// ---- POUs/HydraulicsControl.TcPOU
PROGRAM HydraulicsControl
VAR_INPUT
	// start the hydraulics
	enable:		BOOL := FALSE;
	// reset any hydraulics error
	reset: 		BOOL;
	// manual override to start the suction pump
	suction_manual:	BOOL;
	//manual override to stop the pump
	pump_manual_stop: BOOL;
END_VAR
VAR_OUTPUT
	// status of the brake: is the brake open?
	brake_open:			BOOL;
	// is the brake closed?
	brake_closed:		BOOL;
	// pump is running, but the pressure remains low
	pressure_failure:	BOOL;
	// suction was started, but it is not running
	suction_failure:	BOOL;
	// main pump is running but suction has a timeout
	hydraulics_failure:	BOOL;
	main_pump_failure: BOOL;
	// oil is low
	oil_low:			BOOL;
	// oil is high (unused?)
	oil_high:			BOOL;
	// oil pressure is 25 bars
	oil_pressure_OK:	BOOL;
	// oil is on reserve
	oil_warning:		BOOL;
	// oil filter is dirty
	oil_filter_dirty:	BOOL;
	// oil is below 10°C
	oil_cold:			BOOL;
	// oil is above 50°C
	oil_hot:			BOOL;
	// main pump is running
	pump_running:		BOOL;
	// suction pump is running
	suction_running :	BOOL := FALSE;
	// error condition
	error: 				BOOL;
END_VAR
VAR
	// command to open the brake
	iopen_brake:	BOOL := FALSE;
	// command to open the brake
	iclose_brake: BOOL;
	// monitors the pressure of the pump is running
	pressure_watchdog:	TON;
	// monitors the activation of the suction pump
	suction_watchdog: TON;
	// monitors the activation of the main pump
	main_pump_watchdog:	TON;
	// watch the hydraulics and suction pumps
	hydraulics_watchdog: TON;
	// represents the state of the main pump
	oil_pump_state:		RS;
	// represents the state of the brake
	brake_state: 		RS;
	// wait for the brake to open after pressure has been established
	brake_open_delay:	TON;
	// report brake opend after a short delay
	brake_opened_delay:	TON;
	// error state (set dominant)
	error_state:	SR;
	// trigger for suction pump
	suction_trigger:	SR;
	// timer to shut off hydraulics after break was closed
	hydraulics_off_timer:	TON  := (PT := T#300S);
	off_trigger:	F_TRIG;
	oil_level, last_oil_level:		REAL;
	HydraulicsLog,
	PumpLog,
	ReserveLog,
	oil_low_log,
	FilterLog,
	oil_max_log,
	OverTemperatureLog,
	UnderTemperatureLog,
	SuctionLog,
	HydraulicsFailureLog,
	BrakeClearingWarning,
	BrakeHydraulicsWarning,
	BrakeWarning: FB_EventLog;
	
	// measures the operating cycle of the suction pump
	suction_timer : FB_Timer;
	StatusWord, LastStatus:	UDINT;
END_VAR

(* 
Main control Logic for the Hydraulics system
* power on delay for main pump and suction pump
* start main pump if main control is ready (button pressed or remote)
* start suction pump if maximum in pan is reached
* suction pump runs for 60 seconds
* stop main pump if oil is low
* stop main pump if pressure fails for 10 seconds
*)
oil_low := NOT GVL_Hydraulics.oil_low;
oil_high := NOT GVL_Hydraulics.oil_high;
oil_warning := GVL_Hydraulics.oil_reserve;
oil_pressure_OK := GVL_Hydraulics.oil_pressure_OK;
oil_filter_dirty := NOT GVL_Hydraulics.oilfilter_dirty;
oil_cold := NOT GVL_Hydraulics.oil_undertemperature;
oil_hot := GVL_Hydraulics.oil_overtemperature;
oil_level := F_YREAL(GVL_Hydraulics.oil_level, 0, 16383, 0.0, 5.0);
pump_running := GVL_Hydraulics.pump_running;
suction_running := GVL_Hydraulics.suction_running;

error_state(SET1 := pressure_failure OR	suction_failure OR hydraulics_failure OR oil_low OR main_pump_failure,
			RESET := reset,
			Q1 => error);
// clear reset, if no error present

IF NOT error THEN
	reset := FALSE;
END_IF

oil_pump_state(SET := enable,
				RESET1 := NOT enable OR error OR pump_manual_stop OR GVL_Hydraulics.oilpan_maximum);

GVL_Hydraulics.oil_pump_enable := oil_pump_state.Q1;

(* This section controls the hydraulic brake responsible for azimuth and elevation. 
Especially the elevation is imbalanced if not in the position control loop. 
The brake must only be opened, if the elevation drive is activated concurrently.
*)


// close the brake if the pump is not running	
IF iclose_brake OR NOT pump_running THEN 
	iopen_brake := FALSE;
END_IF

// wait for pressure to build up (hack for oil_pressure_ok)
brake_open_delay(IN := pump_running AND oil_pressure_OK,
				PT := T#3S);
		
brake_state(SET := brake_open_delay.Q AND iopen_brake AND MAIN.brake_clearing,
			RESET1 := GVL_Telescope.azimut_limit_switch 
					  OR iclose_brake 
					  OR NOT pump_running
					  OR NOT MAIN.brake_clearing,
			Q1 => GVL_Telescope.brake_azimuth_eve);

// signal that the brake is open after one second
brake_opened_delay(	IN :=brake_state.Q1, 
					PT := T#1000MS,
					Q => brake_open);

brake_closed := NOT brake_open;
IF brake_closed THEN
	iclose_brake := FALSE;
END_IF
// turn off the hydraulics if the brake is closed and the pump is still running
hydraulics_off_timer(IN := brake_closed AND enable );
off_trigger(CLK := hydraulics_off_timer.Q);

IF hydraulics_off_timer.Q THEN
	enable := FALSE;
END_IF

(* This is the end of the brake control section *)

suction_trigger(SET1 := GVL_Hydraulics.oilpan_maximum OR oil_level>3.7,
				RESET := oil_level<3.0);
GVL_Hydraulics.oil_suction_enable := suction_trigger.Q1 OR suction_manual;					
suction_watchdog(IN := GVL_Hydraulics.oil_suction_enable AND NOT suction_running,
					PT := T#15S,
					Q => suction_failure);
					
pressure_watchdog(IN := GVL_Hydraulics.oil_pump_enable AND 
						NOT oil_pressure_OK,
					PT := T#30S,
				  Q => pressure_failure);
hydraulics_watchdog(IN := pump_running AND NOT suction_running,
						PT := T#140S,
						Q => hydraulics_failure);

main_pump_watchdog(IN := GVL_Hydraulics.oil_pump_enable AND NOT pump_running,
					PT := T#10S,
					Q => main_pump_failure);

StatusWord.0 := oil_low;
StatusWord.1 := oil_high;
StatusWord.2 := oil_warning;
StatusWord.3 := oil_pressure_OK;
StatusWord.4 := oil_filter_dirty;
StatusWord.5 := oil_cold;
StatusWord.6 := oil_hot;
StatusWord.7 := brake_open;
StatusWord.8 := GVL_Main.brake_clearing;
StatusWord.9 := pump_running;
StatusWord.10 := suction_running;
StatusWord.11 := GVL_Hydraulics.oilpan_maximum;
StatusWord.12 := GVL_Hydraulics.oil_pump_enable;
StatusWord.13 := GVL_Hydraulics.oil_suction_enable;
IF ABS(last_oil_level - oil_level) > 0.02 THEN
	StatusWord.15 := TRUE;
	last_oil_level := oil_level;
ELSE
	StatusWord.15 := FALSE;
END_IF

IF StatusWord<>LastStatus THEN // publish new payload every second
	LastStatus := StatusWord;
	MAIN.MQTTClient.Publish('hydraulics', 'base', 'OilLow',			BOOL_TO_STRING(oil_low));
	MAIN.MQTTClient.Publish('hydraulics', 'base', 'OilHigh',		BOOL_TO_STRING(oil_high));
	MAIN.MQTTClient.Publish('hydraulics', 'base', 'OilMaximum',		BOOL_TO_STRING(GVL_Hydraulics.oilpan_maximum));
	MAIN.MQTTClient.Publish('hydraulics', 'base', 'OilReserve',		BOOL_TO_STRING(oil_warning));
	MAIN.MQTTClient.Publish('hydraulics', 'base', 'OilPressureOK', 	BOOL_TO_STRING(oil_pressure_OK));
	MAIN.MQTTClient.Publish('hydraulics', 'base', 'OilFilterDirty',	BOOL_TO_STRING(oil_filter_dirty));
	MAIN.MQTTClient.Publish('hydraulics', 'base', 'OilCold',		BOOL_TO_STRING(oil_cold));
	MAIN.MQTTClient.Publish('hydraulics', 'base', 'OilHot',			BOOL_TO_STRING(oil_Hot));
	MAIN.MQTTClient.Publish('hydraulics', 'base', 'BrakeOpen',		BOOL_TO_STRING(brake_open));
	MAIN.MQTTClient.Publish('hydraulics', 'base', 'BrakeClearing',	BOOL_TO_STRING(GVL_Main.brake_clearing));
	MAIN.MQTTClient.Publish('hydraulics', 'base', 'PumpRunning',	BOOL_TO_STRING(pump_running));
	MAIN.MQTTClient.Publish('hydraulics', 'base', 'SuctionRunning',	BOOL_TO_STRING(suction_running));
	MAIN.MQTTClient.Publish('hydraulics', 'base', 'OilLevel',		REAL_TO_STRING(oil_level));
	MAIN.MQTTClient.Publish('hydraulics', 'base', 'StatusWord',		UDINT_TO_STRING(StatusWord));
END_IF


				  				  
HydraulicsLog(Trigger := pressure_failure OR main_pump_failure,
				Level := ADSLOG_MSGTYPE_ERROR,
				FormatString := 'Main hydraulics pump / pressure: %s',
				OnMessage := 'FAILURE',
				OffMessage := 'OK',
				OffLevel := ADSLOG_MSGTYPE_HINT);

PumpLog(Trigger := pump_running,
				Level := ADSLOG_MSGTYPE_HINT,
				FormatString := 'Main hydraulics pump: %s',
				OnMessage := 'START',
				OffMessage := 'STOP',
				OffLevel := ADSLOG_MSGTYPE_HINT);
	
ReserveLog(Trigger := oil_warning,
			Level := ADSLOG_MSGTYPE_WARN,
			FormatString := 'oil reserve: %s',
			OnMessage := 'LOW',
			OffMessage := 'OK',
			OffLevel := ADSLOG_MSGTYPE_HINT);

oil_low_log(Trigger := oil_low,
				Level := ADSLOG_MSGTYPE_ERROR,
				FormatString := 'oil level: %s',
				OnMessage := 'LOW',
				OffMessage := 'OK',
				OffLevel := ADSLOG_MSGTYPE_HINT);

oil_max_log(Trigger := GVL_Hydraulics.oilpan_maximum,
				Level := ADSLOG_MSGTYPE_ERROR,
				FormatString := 'oil level: %s',
				OnMessage := 'MAXIMUM',
				OffMessage := 'OK',
				OffLevel := ADSLOG_MSGTYPE_HINT);	
				
FilterLog(Trigger := oil_filter_dirty,
				Level := ADSLOG_MSGTYPE_WARN,
				FormatString := 'Hydraulics Filter is %s',
				OnMessage := 'dirty.');

OverTemperatureLog(Trigger := oil_hot,
				Level := ADSLOG_MSGTYPE_WARN,
				FormatString := 'Hydraulics Temperature is %s',
				OnMessage := 'high.');
				
UnderTemperatureLog(Trigger := oil_cold,
				Level := ADSLOG_MSGTYPE_WARN,
				FormatString := 'Hydraulics Temperature is %s',
				OnMessage := 'low.');

SuctionLog(Trigger := suction_failure,
				Level := ADSLOG_MSGTYPE_ERROR,
				FormatString := 'suction pump: %s',
				OnMessage := 'FAILURE',
				OffMessage := 'OK',
				OffLevel := ADSLOG_MSGTYPE_HINT);

HydraulicsFailureLog(Trigger := hydraulics_failure,
				Level := ADSLOG_MSGTYPE_ERROR,
				FormatString := 'suction pump while running main pump: %s',
				OnMessage := 'FAILURE',
				OffMessage := 'OK',
				OffLevel := ADSLOG_MSGTYPE_HINT);
				
BrakeClearingWarning(Trigger := NOT Main.brake_clearing AND iopen_brake,
				Level := ADSLOG_MSGTYPE_WARN,
				FormatString := '%s',
				OnMessage := 'Cannot open brake without brake clearing.');

BrakeWarning(	Trigger := brake_open,
				Level := ADSLOG_MSGTYPE_WARN,
				FormatString := '%s',
				OnMessage := 'Brake is open.',
				OffMessage := 'Brake is closed.');

BrakeHydraulicsWarning(Trigger := NOT enable AND iopen_brake,
				Level := ADSLOG_MSGTYPE_WARN,
				FormatString := '%s',
				OnMessage := 'Cannot open brake without running hydraulics.');

METHOD close_brake : BOOL
VAR_INPUT
END_VAR
// close the brake
iclose_brake := TRUE;

RETURN(brake_closed);
END_METHOD

METHOD open_brake : BOOL
VAR_INPUT
END_VAR
// start the pump
enable := TRUE;
// open the brake
IF oil_pressure_OK THEN
	iopen_brake := TRUE;
END_IF;
RETURN(brake_open);
END_METHOD

END_PROGRAM

// ---- POUs/Functions/F_YREAL.TcPOU
FUNCTION F_YREAL : REAL
VAR_INPUT
	fX:		LREAL;
	fXmin:	REAL := 0.0;
	fXmax:	REAL := 32767.0;
	fYmin, fYmax:	REAL;
END_VAR
VAR
	fgain,
	foffset:	LREAL;
END_VAR

(*
y = mx+b

		    delta X	  fYmax - fYmin
m = fgain = ------- = -------------
			delta Y	  fXmax - fXmin
			
b = foffset = y - m*x = y - fgain*x
					  = fYmin - fgain * fXmin
*)

// y = fgain * x + foffset

IF (fXmax - fXmin) <> 0 THEN

	// Berechnung der Steigung
	fgain := (fYmax - fYmin) / (fXmax - fXmin);
	
	// Berechnung des Offsets
	foffset := fYmin - (fgain * fXmin);
	
	// Berechnung von F_Y

	F_YREAL := LREAL_TO_REAL(fgain * fX + foffset);
	F_YREAL := LIMIT(fYmin, F_YREAL, fYMAX);
END_IF

END_FUNCTION

// ---- POUs/AzimuthElevationControl.TcPOU
PROGRAM AzimuthElevationControl
VAR_INPUT
	// enable the axis and its position control loop
	Enable:		BOOL;
	// reset the axis
	Reset: 		BOOL;
	// decrease azimuth
	left:		BOOL;
	// increase azimuth
	right: 		BOOL;
	// Move azimuth to given position
	MoveAxis:	BOOL;
	// Home the axis
	HomeAxis:	BOOL;
	// enable tracking
	Tracking:	BOOL;
	// position to move the axis to
	position: 	LREAL;
	// set the Velocity of the axis
	velocity:	LREAL;
	// stop the Axis
	StopAxis:	BOOL;
	// diagnostic reset
	bSoEReset:	BOOL;
END_VAR
VAR_OUTPUT
	// error state of the axis
	error: 			BOOL;
	// error ID of the axis
	ErrorID:		UDINT;
	// actual_position of the axis
	act_position:	LREAL;
	// is the axis calibrated
	calibrated:		BOOL;
	// drive is ready
	ready:			BOOL;
	// time to reach target position
	slewtime:		LREAL;
END_VAR
VAR
	AzimuthAxis:		FB_Axis2;
	AzimuthCalibration: MC_SetPosition;
	//fbSoEReset:			FB_SoEReset;
	AzimuthAxisEvent: 	FB_EventLog;
	AzimuthDiagnosticEvent: 	FB_EventLog;
	// delay until commutator angle is measured
	readydelay:			TON;
	HomeDelay:			FB_TONTP;
	TorqueError:		TON := (PT := T#3S);
	azimuth_torque: 	REAL;
	TorqueWarning:		FB_EventLog;
	CalibrationEvent:	FB_Eventlog;
	ReadParameter:		MC_ReadParameter;
	getlastposition:	BOOL := TRUE;
	azimuth_rest_timer:	TON;
	azimuth_at_rest:	BOOL;
	fbSoEReset: 		FB_SoEReset;
	DiagnosticError:	BOOL;
END_VAR
VAR CONSTANT
	// reference position for homing
	// homing_position:		LREAL := 439.0; // was 442 - -21.21 = 463.21; 463 + 24 = 439
	// current position of the calibration cam encoder zero index. Apply an offset here if necessary
	calibration_position:	LREAL :=  208.4983;//208.6273; //208.6073; // 208.7122869;//207.0092; // 208.2342; 
END_VAR
VAR PERSISTENT
	last_position:	LREAL := -1.0;
END_VAR

(* Azimuth Axis control section
Power must be on and brake must be open for the axis to operate
*)

// generate the ready signal after enabling the drive
readydelay(IN :=  AzimuthAxis.Enable, PT := T#3000MS, Q=> ready);

// limit the input position angle
position := LIMIT(0.0, position, 450.0);

// conduct the calibrated signal
calibrated := AzimuthAxis.Calibrated;

IF Calibrated OR Error THEN
	HomeAxis := FALSE;
	getlastposition := FALSE;
END_IF
	
IF HomeAxis THEN
	position := calibration_position;
END_IF

IF HomeDelay.Q THEN
	position := calibration_position;
	MoveAxis := TRUE;
END_IF

// perform a recalibration on the last known position
AzimuthCalibration(
	Axis := GVL_Telescope.AzimuthAxisRef,
	Execute := getlastposition AND last_position>=0.0 AND NOT Calibrated,
	Position := last_position);

IF AzimuthCalibration.Done THEN
	getlastposition := FALSE;
END_IF

IF Calibrated THEN
	last_position := act_position;
END_IF

// enable the azimuth if not moved by the power chain. Sorry for the hack
azimuth_rest_timer(IN := HydraulicsControl.brake_open AND 
				(ABS(GVL_Telescope.AzimuthAxisRef.NcToPlc.ActVelo) < 0.01), PT := T#2S);
// if azimuth at rest or calibrated, allow enabling the azimuth
IF azimuth_rest_timer.Q or calibrated THEN
	azimuth_at_rest := TRUE;
ELSIF HydraulicsControl.brake_closed THEN
	azimuth_at_rest := FALSE;
END_IF
	
// deactivate limit switches on homing
MC_SetAcceptBlockedDriveSignal(
	Axis := GVL_Telescope.AzimuthAxisRef, 
	Enable := HomeAxis);

AzimuthAxis(	
	Enable := 			enable AND azimuth_at_rest AND NOT GVL_Telescope.azimut_limit_switch,
	Reset := 			reset,
	MoveAxis :=			MoveAxis,
	HomeAxis := 		HomeAxis,
	StopAxis :=			StopAxis,
	Tracking :=			Tracking,
	Position := 		position, 
	Velocity :=			velocity,
	Enable_Positive := 	GVL_Telescope.Azimuth_inputs.1 OR HomeAxis,
	Enable_Negative := 	GVL_Telescope.Azimuth_inputs.0,
	Jog_Forward :=		right,
	Jog_Backwards := 	left,
	bCalibrationCam :=	NOT GVL_Telescope.Azimuth_inputs.1,
	ActualPosition => 	act_position,
	Error => 			error,
	ErrorID => 			ErrorID,
	AxisRef :=			GVL_Telescope.AzimuthAxisRef);

IF bSoEReset THEN
	last_position := -1.0;
	fbSoEReset(
		Axis := GVL_Telescope.AzimuthAxisRef,
		Execute := TRUE,
		Timeout := DEFAULT_ADS_TIMEOUT);
 	IF fbSoEReset.Busy THEN
		fbSoEReset(Axis := GVL_Telescope.AzimuthAxisRef, Execute := FALSE);
	ELSE
		bSoEReset := FALSE;
		Reset := TRUE;
	END_IF
END_IF 

IF AzimuthAxis.MoveDone THEN
	MoveAxis := FALSE;
END_IF

IF AzimuthAxis.HomeDone THEN
	HomeAxis := FALSE;
END_IF
	
IF AzimuthAxis.ResetDone THEN
	reset := FALSE;
END_IF

IF AzimuthAxis.StopDone THEN
	StopAxis := FALSE;
END_IF
DiagnosticError := FALSE;
IF GVL_Telescope.Azimuth_diagnostic < 16#D012 AND GVL_Telescope.Azimuth_diagnostic > 16#D014 THEN
	DiagnosticError :=TRUE;
	ErrorID := GVL_Telescope.Azimuth_diagnostic;
END_IF

ReadParameter(	Axis := GVL_Telescope.AzimuthAxisRef, Enable := AzimuthAxis.InMotion, 
				ParameterNumber := MC_AxisParameter.AxisRemainingTimeToGo, 
				ReadMode := E_ReadMode.READMODE_CYCLIC);
IF ReadParameter.Valid THEN
	slewtime := ReadParameter.Value;
END_IF

azimuth_torque := GVL_Telescope.Azimuth_torque / 10.0;
TorqueError(IN := ABS(azimuth_torque) > 50.0);


AzimuthAxisEvent(	
	Trigger := 		Error, 
	Level := 		ADSLOG_MSGTYPE_ERROR,
	FormatString :=	'Azimuth Axis Error: %s',
	OnMessage := 	NCError_TO_STRING(ErrorID));
	
AzimuthDiagnosticEvent(	
	Trigger := 		DiagnosticError,
	Level := 		ADSLOG_MSGTYPE_ERROR,
	FormatString :=	'Azimuth Axis Diagnostic Error: %s',
	OnMessage := 	NCError_TO_STRING(GVL_Telescope.Azimuth_diagnostic));
	
TorqueWarning(	
	Trigger := 		TorqueError.Q, 
	Level := 		ADSLOG_MSGTYPE_WARN,
	FormatString :=	'%s',
	OnMessage := 	'Azimuth torque is high.');
	
CalibrationEvent(
	Trigger := 		Calibrated, 
	Level := 		ADSLOG_MSGTYPE_HINT,
	FormatString :=	'%s',
	OnMessage := 	'Azimuth axis is calibrated.');

END_PROGRAM

// ---- POUs/FunctionBlocks/FB_TONTP.TcPOU
FUNCTION_BLOCK FB_TONTP
VAR_INPUT
	IN :	BOOL;
	 PT1:	TIME := T#1000MS;
	 PT2:	TIME := T#1000MS;
END_VAR
VAR_OUTPUT
	Q:	BOOL;
END_VAR
VAR
	ton:	TON;
	tp:		TP;
END_VAR

ton(IN := IN, PT := PT1);
tp(IN := ton.Q, PT := PT2, Q => Q);

END_FUNCTION_BLOCK

// ---- POUs/FilterWheelControl.TcPOU
PROGRAM FilterWheelControl
VAR_INPUT
	// enable the axis
	Enable:				BOOL;
	// reset the axis(-error)
	Reset:				BOOL;
	// move counter-clockwise
	left:				BOOL;
	// move clockwise
	right:				BOOL;
	// TRUE, if the filter is in position and wheel has come to rest
	Ready:				BOOL;
	// filter position
	filter_position: 	USINT;
	// move to given position
	MoveAxis: 			BOOL;
	// calibrate the axis
	HomeAxis:			BOOL;
END_VAR
VAR_OUTPUT
	// is true if an error occurred
	error: 				BOOL;
	// number of current axis error
	ErrorID:			UDINT;
	act_position:		LREAL;
	// axis has been calibrated
	Calibrated :		BOOL;
END_VAR
VAR
	FilterWheelAxis:	FB_Axis2;
	// axis position to set to with `MoveAxis`
	position:			LREAL;
	// current filter determined from the axis position
	actual_filter:		USINT;
	FilterWheelEvent:	FB_EventLog;
	CalibratedEvent:	FB_EventLog;
	FilterReadyEvent:	FB_Eventlog;
	Calibration1Event:	FB_Eventlog;
	Calibration2Event:	FB_Eventlog;
	
	// last known filter position
	last_filter_position:	USINT;
	HomingMode:			MC_HomingMode := MC_HomingMode.MC_ForceCalibration;
	MQTTTimer : 		TON := (PT:=T#5S);
	CalibrationTrigger1:	R_TRIG;
	CalibrationTrigger2:	F_TRIG;
END_VAR
VAR CONSTANT
	// total number of filters in the filter wheel
	filters:			USINT := 24;
	// current position of the calibration cam. Apply an offset here if necessary
	calibration_position:	LREAL := 1.8;
END_VAR

(* This program controls the filter wheel. 
The current optical filter is selected through `filter_position`.
The number of filters is hard coded to 24.

*)

// limit desired filter_position to [0...filters-1]
filter_position := filter_position MOD filters;
// calculate the actual filter position
actual_filter := LREAL_TO_USINT((360.0 - act_position) * filters / 360.0) MOD filters;

Ready := (filter_position = actual_filter) AND (FilterWheelAxis.Standstill OR NOT Enable);
IF Pendantcontrol.telescope_mode = E_TelescopeMode.automatic THEN
	IF FilterWheelAxis.Calibrated THEN
		// if we are on automatic mode then position the filterwheel
		position := MODABS(360.0 - 360.0 * WORD_TO_LREAL(filter_position) / WORD_TO_LREAL(filters), 360.0);
		IF filter_position <> actual_filter THEN
			IF FilterWheelAxis.Ready THEN
				MoveAxis := TRUE;	
			ELSE
				Enable := TRUE;
			END_IF
		END_IF
		IF FilterWheelAxis.MoveDone THEN
			Enable := FALSE;
		END_IF
	ELSE
		IF FilterWheelAxis.Ready THEN
			HomeAxis := TRUE;
		END_IF
	END_IF
END_IF
IF HomeAxis THEN
	IF HomingMode = MC_HomingMode.MC_DefaultHoming THEN
		position := calibration_position;
		filter_position := 0;	
	END_IF
END_IF

Calibrated := FilterWheelAxis.Calibrated;

FilterWheelAxis(
	Enable := 			Enable,
	Reset := 			Reset,
	MoveAxis :=			MoveAxis,
	HomeAxis :=			HomeAxis,
	HomingMode :=		HomingMode,
	Position := 		position, 
	Velocity :=			30.0, //60.0,
	Enable_Positive :=  TRUE,
	Enable_Negative := 	TRUE,
	Jog_Forward :=		left,
	Jog_Backwards := 	right,
	bCalibrationCam :=	NOT GVL_FilterWheel.bCalibrationCam,
	isModuloAxis :=		TRUE,
	ActualPosition => 	act_position,
	Error => 			error,
	ErrorID => 			ErrorID,
	AxisRef :=			GVL_FilterWheel.FilterWheel_AxisRef);

IF FilterWheelAxis.MoveDone THEN
	MoveAxis := FALSE;
END_IF

IF FilterWheelAxis.HomeDone THEN
	HomeAxis := FALSE;
	Enable := FALSE;
END_IF
	
IF FilterWheelAxis.ResetDone THEN
	reset := FALSE;
END_IF

CalibrationTrigger1(CLK := GVL_FilterWheel.bCalibrationCam);
CalibrationTrigger2(CLK := GVL_FilterWheel.bCalibrationCam);


MQTTTimer(IN:=TRUE);
IF actual_filter <> last_filter_position OR MQTTTimer.Q THEN
	MAIN.MQTTClient.Publish('telescope', 'dome', 'FilterPosition', WORD_TO_STRING(actual_filter));
	MAIN.MQTTClient.Publish('telescope', 'dome', 'FilterWheelReady', BOOL_TO_STRING(Ready));
	last_filter_position := actual_filter;
	MQTTTimer(IN:=FALSE);
END_IF

FilterWheelEvent(	
	Trigger := 		Error, 
	Level := 		ADSLOG_MSGTYPE_ERROR,
	FormatString :=	'Filter Wheel Axis Error: %s',
	OnMessage := 	NCError_TO_STRING(ErrorID),
	OffMEssage := 	'OK',
	OffLevel := 	ADSLOG_MSGTYPE_HINT);
	
CalibratedEvent(
	Trigger :=		Calibrated,
	Level := 		ADSLOG_MSGTYPE_HINT,
	FormatString :=	'%s',
	OnMessage := 	'Filter wheel is calibrated.');
	
FilterReadyEvent(
	Trigger :=		(filter_position = actual_filter) AND Calibrated,
	Level := 		ADSLOG_MSGTYPE_HINT,
	FormatString :=	'Filter position %s is ready.',
	OnMessage := 	WORD_TO_STRING(actual_filter));
	
Calibration1Event(
	Trigger :=	CalibrationTrigger1.Q,
	Level := 		ADSLOG_MSGTYPE_HINT,
	FormatString :=	'Calibration raising signal triggered at position: %s',
	OnMessage := 	LREAL_TO_STRING(act_position));

Calibration2Event(
	Trigger :=	CalibrationTrigger2.Q,
	Level := 		ADSLOG_MSGTYPE_HINT,
	FormatString :=	'Calibration falling signal triggered at position: %s',
	OnMessage := 	LREAL_TO_STRING(act_position));

END_PROGRAM

// ---- POUs/TelescopeControl.TcPOU
PROGRAM TelescopeControl
VAR_INPUT
(*
TCS interface section
see https://gitlab.aip.de/bmk10k/telescope_firmware/snippets/5
*)
	
	// boolean, true: Power on, false: power off
	power: 		BOOL;
	// boolean, true: go to home position, unset track/goto if active
	gohome: 	BOOL;
	// boolean, true: go into park position, ready to stow telescope, unset track/goto
	park: 		BOOL;
	// boolean, TRUE: MOVE telescope TO last ra/de AND start tracking. Set 'goto' TO FALSE, IF TRUE. FALSE: Stop tracking as soon as possible
	track: 		BOOL;
	// boolean, TRUE: MOVE telescope TO tau/de AND stop there. Set track TO FALSE, IF TRUE. FALSE: no effect.)
	goto:		BOOL;	
	// move the telescope to a given az-alt position
	slew:		BOOL;
	// boolean, TRUE: Stop motion OF telescope immediately, set goto AND track TO FALSE. FALSE: Allow motion OF telescope again via track/goto).
	stop:		BOOL;	
	// initiates reset on all axis
	reset:		BOOL;
	// automatic tracking after goto
	autotrack:	BOOL := TRUE;
	// apparent right ascension, degrees, double
	rightascension:		LREAL := (4.0 + 35.0/60.0 + 54.09/3600.0) *15.0;	
	// apparent declination, degrees, double
	declination: 		LREAL := 16.0 + 30.0/60.0 + 25.4/3600.0;
	// desired elevation of the telescope pointing 
	elevation:	LREAL := 45.0;
	// desired azimut of the telescope pointing 
	azimuth:	LREAL := 320.0;
	// absolute offset for elevation
	elevation_offset:	LREAL := 0.0;
	// absolute offset for azimuth
	azimuth_offset : 	LREAL := 0.0;
	// absolute offset for time
	time_offset: 		LREAL := 0.0;
	// offset for the de-rotator
	derotator_offset:	LREAL := 0.0;
	// Nasmyth port 1 or 2
	Nasmyth_port: 		USINT;
END_VAR
VAR
	// actual command from the TCS
	TCS_command: 	E_TCSCommand;
	// current Julian Date calculated from system time
	jd:				LREAL;
	// image derotation
	derotation_calc:	LREAL;
	// local siderial time calculated from Julian date
	lst:			LREAL;
	// elevation calulated when ra and dec are set by TCS
	elevation_calc:	LREAL; 
	// azimuth calulated when ra and dec are set by TCS
	azimuth_calc:	LREAL;
	// right ascension calulated when azimuth and elevation are set by TCS
	rightascension_calc:	LREAL;
	// declination calulated when azimuth and elevation are set by TCS
	declination_calc:		LREAL;
	// hour angle
	Hourangle_calc: LREAL;
	// precise astronomical	time
	fbTime: FB_AstroClock;
	
	eq2hor2:	FB_EQ2HOR2;
	hor2eq:		FB_HOR2EQ;
	
	// triggers power-failure event
	powerfailure: 	BOOL;
	// triggers power warning
	poweronwarning:	TP;
	// power on timeout
	power_timeout:	TON;
	// command timeout
	command_timeout:	TON;
	// tracking delay
	tracking_delay:	TON;
	// telescope is parked
	isparked:		BOOL;
	TCSpowerEvent,
	TCSgohomeEvent,
	TCSparkEvent,
	TCSgotoEvent,
	TCStrackEvent,
	TCSstopEvent,
	AltitudeEvent,
	TCSreadyEvent,
	TCSCTOEvent: FB_Eventlog;
	MQTTTimer : TON := (PT:=T#5S);
	// rotational velocity of the derotator
	DerotatorVelocity: LREAL;
	// rotational velocity of the elevation
	ElevationVelocity: LREAL;
	// rotational velocity of the elevation
	AzimuthVelocity: LREAL;
	// sign of derotation
	derotatation_sign: LREAL := 1.0;
	StatusWord, LastStatus:	UDINT;
END_VAR
VAR_OUTPUT
	//		TRUE, IF telescope can be operated
	ready:		BOOL; 
	// indicates an error on one of the components
	error:		BOOL;	
	//error id of axis
	errorid:	UDINT;	
	//TRUE, IF telescope is in fast-MOVE phase (includes pole-swap)
	sliding:	BOOL;	
	//TRUE, IF telescope is on tracking position AND currently tracking.
	tracking:	BOOL;	
	//TRUE, IF telescope is AT rest.
	stopped:	BOOL;	
	// true position of the elevation
	elevation_current:	LREAL;
	// true position of the azimuth
	azimuth_current:	LREAL;
	// true position of the de-rotator
	derotator_current:	LREAL;
	//	(time in sec. to reach the goto/track position)
	slewtime:			LREAL; 
	// True: telescope is calibrated
	homed:				BOOL;
	// telescope does not accept further commands
	busy:				BOOL;
END_VAR
VAR CONSTANT
// STELLA1
	// telescope site longitude, source: Google 
	longitude: 		LREAL := -16.50926; //13.101867;
	// telescope site latitude, source: Google
	latitude: 		LREAL := 28.30120; //52.404940;
	// telescope site height above sea level: estimated
	altitude: 		LREAL := 2390.0;
	elevation_park: LREAL := 60.0;
	azimuth_park: 	LREAL := 359.999;
	derotator_park: LREAL := 229.85;

	elevation_home: LREAL := 55.0;
	azimuth_home: 	LREAL := 180.0;
END_VAR
VAR PERSISTENT
	// azimuth axis offset/misalignment north-south
	AN_E:	LREAL;
	// azimuth axis offset/misalignment east-west
	AE_E:	LREAL;
	// gravitational flexure correction at the horizon
	TF:		LREAL;
	// collimation error of the electromagnetic axis
	BNP:	LREAL;
	// azimuth axis offset/misalignment north-south
	AN_A:	LREAL;
	// azimuth axis offset/misalignment east-west,
	AE_A:	LREAL;
	// Non-perpendicularity between the mount azimuth and elevation axes
	NPAE:	LREAL;
END_VAR

TelescopeAuxiliary();

// get the system time
fbTime();
jd := DateTime2JD(fbTime.time_RTCEX2);
lst := CT2LST(longitude, jd);
// set reset state either by hardware (key pressed) or by software (set by e.g. tcs)
IF GVL_Main.reset_switch THEN
	reset := TRUE;
END_IF


IF ElevationControl.error THEN
	errorid := ElevationControl.ErrorID;
	ElevationControl.reset := reset;
ELSIF AzimuthElevationControl.error THEN
	errorid := AzimuthElevationControl.ErrorID;
	AzimuthElevationControl.Reset := reset;
ELSIF FilterWheelControl.Error THEN
	errorid := FilterWheelControl.ErrorID;
	FilterWheelControl.Reset := reset;
ELSIF Focuscontrol.Error THEN
	errorid := Focuscontrol.ErrorID;
	FocusControl.reset := reset;
ELSIF DerotatorControl.Error THEN
	errorid := DerotatorControl.ErrorID;
	DerotatorControl.reset := reset;
END_IF

error := ElevationControl.error OR 
		 AzimuthElevationControl.error OR
		 FilterWheelControl.Error OR
		 Focuscontrol.Error OR
		 DerotatorControl.Error;

slewtime := MAX(MAX(ElevationControl.slewtime, AzimuthElevationControl.slewtime), DerotatorControl.slewtime);
			
IF error THEN
	gohome := 	FALSE;
	track := 	FALSE;
	goto := 	FALSE;
	slew := 	FALSE;
ELSE
	errorid := 0;
END_IF

IF ElevationControl.error THEN
	ElevationControl.enable := FALSE;
	AzimuthElevationControl.enable := FALSE;
	HydraulicsControl.close_brake();
END_IF

eq2hor2(alpha := rightascension,
	delta := declination,
	lon := longitude,
	lat := latitude,
	JD := jd + time_offset,
	alt => elevation_calc,
	az => azimuth_calc,
	ha => hourangle_calc);

// apply pointing model
elevation_calc := elevation_calc + PointingModelElevation(azimuth_calc, elevation_calc, elevation_offset, AN_E, AE_E, TF);
azimuth_calc := azimuth_calc + PointingModelAzimuth(azimuth_calc, elevation_calc, azimuth_offset, BNP, AN_A, AE_A, NPAE);
// calculate derotator position 
derotation_calc := F_DerotatorPosition2(azimuth_calc, elevation_calc, declination_calc, latitude, derotatation_sign)  + derotator_offset;
// calculate velocities
DerotatorVelocity := F_Derotatorvelocity(elevation_calc, azimuth_calc, latitude);
ElevationVelocity := F_Elevationvelocity(azimuth_calc, latitude);
AzimuthVelocity := F_Azimuthvelocity(elevation_calc, azimuth_calc, latitude);

IF (azimuth_calc > 310.0 AND AzimuthVelocity > 0.0) OR (azimuth_calc > 440.0) THEN
	azimuth_calc := azimuth_calc - 360.0;
ELSIF (azimuth_calc < 80.0 AND AzimuthVelocity < 0.0) OR (azimuth_calc < -50.0) THEN
	azimuth_calc := azimuth_calc + 360.0;
END_IF

IF (derotation_calc > 290.0 AND DerotatorVelocity > 0.0) OR (derotation_calc > 380.0) THEN
	derotation_calc := derotation_calc - 360.0;
ELSIF (derotation_calc < 20.0 AND DerotatorVelocity < 0.0) OR (derotation_calc < -70.0) THEN
	derotation_calc := derotation_calc + 360.0;
END_IF
// get current coordinates	
azimuth_current := AzimuthElevationControl.act_position;
elevation_current := ElevationControl.actual_position;
derotator_current := DerotatorControl.actual_position;

// calculate equatorial coordinates
hor2eq(alt := elevation_current - PointingModelElevation(azimuth_calc, elevation_calc, elevation_offset, AN_E, AE_E, TF), 
		az := azimuth_current - PointingModelAzimuth(azimuth_calc, elevation_calc, azimuth_offset, BNP, AN_A, AE_A, NPAE),
		jd := jd,
		lat := latitude,
		lon := longitude,
		altitude := altitude,
		ra => rightascension_calc,
		dec => declination_calc);		
	
poweronwarning(IN := power OR (NOT ElevationControl.enable AND HydraulicsControl.brake_open), PT := T#250MS);

power_timeout(IN := TCS_command = E_TCSCommand.no_command AND NOT isparked, PT := T#12H);
command_timeout();
IF power_timeout.Q AND NOT isparked THEN
	park := TRUE;
END_IF

IF Nasmyth_port = 1 THEN
	NasmythControl.right := FALSE;
	IF NasmythControl.Nasmyth_left THEN
		NasmythControl.left := FALSE;
		NasmythControl.enable := FALSE;
	ELSE
		NasmythControl.left := TRUE;
		NasmythControl.enable := TRUE;
	END_IF
ELSIF Nasmyth_port = 2 THEN
	NasmythControl.left := FALSE;
    IF NasMythControl.Nasmyth_right THEN
		NasmythControl.right := FALSE;
		NasmythControl.enable := FALSE;
	ELSE
		NasmythControl.right := TRUE;
		NasmythControl.enable := TRUE;
	END_IF
ELSE
	NasmythControl.right := FALSE;
	NasmythControl.left := FALSE;
	NasmythControl.enable := FALSE;	
END_IF
	
		
// set TCS_command according to state variables ordered by precedence
IF power THEN
	TCS_command := E_TCSCommand.poweron;
ELSIF stop THEN
	TCS_command := E_TCSCommand.stop;
	goto := FALSE;
	track := FALSE;
	slew := FALSE;
	gohome := FALSE;
	park := FALSE;
ELSIF park THEN
	goto := FALSE;
	track := FALSE;
	slew := FALSE;
	IF ready AND stopped THEN
		TCS_command := E_TCSCommand.park;
	END_IF
ELSIF gohome THEN
	goto := FALSE;
	track := FALSE;
	slew := FALSE;
	IF ready AND NOT busy AND stopped THEN
		TCS_command := E_TCSCommand.gohome;
	END_IF
ELSIF goto THEN
	track := FALSE;
	slew := FALSE;
	IF ready AND NOT busy THEN
		TCS_command := E_TCSCommand.goto;
	END_IF
ELSIF slew THEN
	goto := FALSE;
	track := FALSE;
	IF ready AND NOT busy THEN
		TCS_command := E_TCSCommand.slew;
	END_IF
ELSIF track THEN
	goto := FALSE;
	slew := FALSE;
	IF ready AND NOT busy THEN
		TCS_command := E_TCSCommand.track;
	END_IF
ELSE
	TCS_command := E_TCSCommand.no_command;
	ElevationControl.MoveAxis := FALSE;
	AzimuthElevationControl.MoveAxis := FALSE;
	DerotatorControl.MoveAxis := FALSE;
	ElevationControl.Tracking := FALSE;
	AzimuthElevationControl.Tracking := FALSE;
	DerotatorControl.Tracking := FALSE;
END_IF

IF TCS_command = E_TCSCommand.poweron THEN
	poweron();
	command_timeout(IN := TCS_command = E_TCSCommand.poweron, PT := T#12H);
	TCSCTOEvent.OnMessage := 'POWER';
ELSIF TCS_command = E_TCSCommand.stop THEN
	stoptelescope();
	command_timeout(IN := TCS_command = E_TCSCommand.stop, PT := T#2S);
	TCSCTOEvent.OnMessage := 'STOP';
ELSIF TCS_command = E_TCSCommand.park THEN
	parktelescope();
	command_timeout(IN := TCS_command = E_TCSCommand.park, PT := T#2M);
	TCSCTOEvent.OnMessage := 'PARK';
ELSIF TCS_command = E_TCSCommand.gohome THEN
	hometelescope();
	command_timeout(IN := TCS_command = E_TCSCommand.gohome, PT := T#2M);
	TCSCTOEvent.OnMessage := 'GOHOME';
ELSIF TCS_command = E_TCSCommand.goto THEN
	gototelescope();
	command_timeout(IN := TCS_command = E_TCSCommand.goto, PT := T#2M);
	TCSCTOEvent.OnMessage := 'GOTO';
ELSIF TCS_command = E_TCSCommand.slew THEN
	slewtelescope();
	command_timeout(IN := TCS_command = E_TCSCommand.slew, PT := T#2M);
	TCSCTOEvent.OnMessage := 'SLEW';
ELSIF TCS_command = E_TCSCommand.track THEN
	tracktelescope();
	command_timeout(IN := TCS_command = E_TCSCommand.track, PT := T#12H);
	TCSCTOEvent.OnMessage := 'TRACK';
ELSE
	// disable command timeout
	command_timeout(IN := FALSE);
	TCSCTOEvent.OnMessage := 'NOCOMMAND';
END_IF
 
sliding := NOT tracking AND (ElevationControl.ElevationAxis.InMotion OR ElevationControl.ElevationAxis.InRamp OR
			AzimuthElevationControl.AzimuthAxis.InMotion OR AzimuthElevationControl.AzimuthAxis.InRamp OR
			DerotatorControl.DerotatorAxis.InMotion OR DerotatorControl.DerotatorAxis.InRamp);

// signal must be stable for 5500MS			
tracking_delay(in := ElevationControl.ElevationAxis.isTracking AND 
			AzimuthElevationControl.AzimuthAxis.isTracking AND
			DerotatorControl.DerotatorAxis.isTracking,PT :=T#5500MS, Q => tracking);
			
stopped :=  (NOT ElevationControl.enable OR ElevationControl.ElevationAxis.StandStill) AND 
			(NOT AzimuthElevationControl.Enable OR AzimuthElevationControl.AzimuthAxis.StandStill) AND
			(NOT DerotatorControl.enable OR DerotatorControl.DerotatorAxis.StandStill);
			
homed := ElevationControl.Calibrated AND
			AzimuthElevationControl.calibrated AND
			FilterWheelControl.Calibrated AND
			FocusControl.Calibrated AND
			DerotatorControl.Calibrated;
			
ready := homed AND 
	CoverControl.isopen AND 
	ElevationControl.enable AND
	AzimuthElevationControl.enable AND
	DerotatorControl.enable AND HydraulicsControl.brake_open AND 
    NOT error;

busy := ElevationControl.ElevationAxis.Busy OR
		AzimuthElevationControl.AzimuthAxis.Busy OR
		DerotatorControl.DerotatorAxis.Busy OR
		FocusControl.FocusAxis.Busy OR
		FilterWheelControl.FilterWheelAxis.Busy;
		
// unset the STOP command if telescope is already stopped
IF stopped THEN
	stop := FALSE;
END_IF
	
IF NOT error THEN
	reset := FALSE;
END_IF

IF SafetyHandling.Emergency_stop THEN
	ElevationControl.enable := FALSE;
	AzimuthElevationControl.enable := FALSE;
	DerotatorControl.enable := FALSE;
END_IF
IF sliding OR track OR tracking THEN
	MQTTTimer.PT := T#1000MS;
ELSE
	MQTTTimer.PT := T#5000MS;
END_IF
MQTTTimer(IN:=TRUE);
IF MQTTTimer.Q THEN // publish new payload every second
	MQTTTimer(IN:=FALSE);

	MAIN.MQTTClient.Publish('telescope', 'dome', 'JulianDate', LREAL_TO_STRING(jd));
	MAIN.MQTTClient.Publish('telescope', 'dome', 'LocalSiderialTime', LREAL_TO_STRING(lst));
	MAIN.MQTTClient.Publish('telescope', 'dome', 'Azimuth', LREAL_TO_STRING(azimuth_current));
	MAIN.MQTTClient.Publish('telescope', 'dome', 'Elevation', LREAL_TO_STRING(elevation_current));
	MAIN.MQTTClient.Publish('telescope', 'dome', 'Derotator', LREAL_TO_STRING(derotator_current));
	MAIN.MQTTClient.Publish('telescope', 'dome', 'HourAngle', LREAL_TO_STRING(hourangle_calc));
	MAIN.MQTTClient.Publish('telescope', 'dome', 'RightAscension', LREAL_TO_STRING(rightascension_calc));
	MAIN.MQTTClient.Publish('telescope', 'dome', 'Declination', LREAL_TO_STRING(declination_calc));
	MAIN.MQTTClient.Publish('telescope', 'dome', 'azimuth_offset', LREAL_TO_STRING(azimuth_offset));
	MAIN.MQTTClient.Publish('telescope', 'dome', 'elevation_offset', LREAL_TO_STRING(elevation_offset));
	MAIN.MQTTClient.Publish('telescope', 'dome', 'derotator_torque', LREAL_TO_STRING(DerotatorControl.derotator_torque));
	MAIN.MQTTClient.Publish('telescope', 'dome', 'elevation_torque', LREAL_TO_STRING(ElevationControl.elevation_torque));
	MAIN.MQTTClient.Publish('telescope', 'dome', 'azimuth_torque', LREAL_TO_STRING(AzimuthElevationControl.azimuth_torque));
	
	MAIN.MQTTClient.Publish('telescope', 'dome', 'errorid',		UDINT_TO_STRING(errorid));
	MAIN.MQTTClient.Publish('telescope', 'dome', 'error',		BOOL_TO_STRING(error));
	MAIN.MQTTClient.Publish('telescope', 'dome', 'ready',		BOOL_TO_STRING(ready));
	MAIN.MQTTClient.Publish('telescope', 'dome', 'busy',		BOOL_TO_STRING(busy));
	MAIN.MQTTClient.Publish('telescope', 'dome', 'sliding',		BOOL_TO_STRING(sliding));
	MAIN.MQTTClient.Publish('telescope', 'dome', 'tracking', 	BOOL_TO_STRING(tracking));
	MAIN.MQTTClient.Publish('telescope', 'dome', 'stopped',		BOOL_TO_STRING(stopped));
	MAIN.MQTTClient.Publish('telescope', 'dome', 'homed',		BOOL_TO_STRING(homed));
END_IF

StatusWord.0 := error;
StatusWord.1 := ready;
StatusWord.2 := sliding;
StatusWord.3 := tracking;
StatusWord.4 := stopped;
StatusWord.5 := homed;
StatusWord.6 := power;
StatusWord.7 := park;
StatusWord.8 := gohome;
StatusWord.9 := track;
StatusWord.10 := goto;
StatusWord.11 := slew;
StatusWord.12 := stop;
StatusWord.13 := busy;

IF StatusWord<>LastStatus THEN // publish new payload every second
	LastStatus := StatusWord;
	MAIN.MQTTClient.Publish('telescope', 'dome', 'error',		BOOL_TO_STRING(error));
	MAIN.MQTTClient.Publish('telescope', 'dome', 'ready',		BOOL_TO_STRING(ready));
	MAIN.MQTTClient.Publish('telescope', 'dome', 'sliding',		BOOL_TO_STRING(sliding));
	MAIN.MQTTClient.Publish('telescope', 'dome', 'tracking', 	BOOL_TO_STRING(tracking));
	MAIN.MQTTClient.Publish('telescope', 'dome', 'stopped',		BOOL_TO_STRING(stopped));
	MAIN.MQTTClient.Publish('telescope', 'dome', 'homed',		BOOL_TO_STRING(homed));
	MAIN.MQTTClient.Publish('telescope', 'dome', 'power',		BOOL_TO_STRING(power));
	MAIN.MQTTClient.Publish('telescope', 'dome', 'park',		BOOL_TO_STRING(park));
	MAIN.MQTTClient.Publish('telescope', 'dome', 'gohome',		BOOL_TO_STRING(gohome));
	MAIN.MQTTClient.Publish('telescope', 'dome', 'track',		BOOL_TO_STRING(track));
	MAIN.MQTTClient.Publish('telescope', 'dome', 'goto',		BOOL_TO_STRING(goto));
	MAIN.MQTTClient.Publish('telescope', 'dome', 'slew',		BOOL_TO_STRING(slew));
	MAIN.MQTTClient.Publish('telescope', 'dome', 'stop',		BOOL_TO_STRING(stop));
	MAIN.MQTTClient.Publish('telescope', 'dome', 'busy',		BOOL_TO_STRING(busy));
END_IF


(* Event function blocks start here. *)
TCSpowerEvent(	Trigger := powerfailure, 
				Level := ADSLOG_MSGTYPE_ERROR,
				FormatString := 'power %s',
				OnMessage := 'Failure',
				OffMessage := 'OK');

TCSgohomeEvent(	Trigger := gohome, 
				Level := ADSLOG_MSGTYPE_HINT,
				FormatString := 'GOHOME %s',
				OnMessage := 'commencing',
				OffMEssage := 'completed');
TCSparkEvent(	Trigger := park, 
				Level := ADSLOG_MSGTYPE_HINT,
				FormatString := 'PARK %s',
				OnMessage := 'commencing',
				OffMEssage := 'completed');
TCSgotoEvent(	Trigger := goto, 
				Level := ADSLOG_MSGTYPE_HINT,
				FormatString := 'GOTO %s',
				OnMessage := 'commencing',
				OffMEssage := 'completed');
TCStrackEvent(	Trigger := track, 
				Level := ADSLOG_MSGTYPE_HINT,
				FormatString := 'TRACK %s',
				OnMessage := 'commencing',
				OffMEssage := 'completed');
TCSstopEvent(	Trigger := stop, 
				Level := ADSLOG_MSGTYPE_WARN,
				FormatString := 'STOP %s',
				OnMessage := 'commencing',
				OffMEssage := 'completed',
				OffLevel := ADSLOG_MSGTYPE_HINT);
AltitudeEvent(	Trigger := power AND elevation_calc<0.0, 
				Level := ADSLOG_MSGTYPE_WARN,
				FormatString := '%s',
				OnMessage := 'Target below horizon',
				OffMEssage := '');
TCSreadyEvent(	Trigger := power AND ready, 
				Level := ADSLOG_MSGTYPE_HINT,
				FormatString := '%s',
				OnMessage := 'STELLA1 startup finished');
TCSCTOEvent(	Trigger := command_timeout.Q, 
				Level := ADSLOG_MSGTYPE_WARN,
				FormatString := 'A timeout occured during %s command!',
				OnMessage := 'NOCOMMAND');

METHOD gototelescope: USINT
VAR_INPUT
END_VAR
VAR
	GoToEvent:	FB_Eventlog;
	command_timeout:	TON;
END_VAR
VAR_STAT
	Stage:		USINT := 0;
	LastStage:	USINT := 101;
END_VAR
gototelescope := Stage;
command_timeout(IN := Stage < 100, PT := T#600S);
IF command_timeout.Q THEN
	error := TRUE;
	errorid := 16#10;
	goto := FALSE;
	Stage := 0;
	RETURN;
END_IF

IF elevation_calc<2.0 THEN
	error := TRUE;
	errorid := 16#15;
	goto := FALSE;
	Stage := 0;
	RETURN;
END_IF

IF reset OR error THEN
	Stage := 0;
	RETURN;
END_IF

CASE Stage OF
	0:	
		IF ready AND NOT busy THEN
			Stage := 25;
		END_IF
	25:	
		ElevationControl.position := elevation_calc;
		AzimuthElevationControl.position := azimuth_calc;
		DerotatorControl.position := derotation_calc;
		DerotatorControl.Velocity := 10.0;
		ElevationControl.velocity := 10.0;
		AzimuthElevationControl.velocity := 10.0;
		
		ElevationControl.MoveAxis := TRUE;
		AzimuthElevationControl.MoveAxis := TRUE;
		DerotatorControl.MoveAxis := TRUE;
		IF ElevationControl.ElevationAxis.Busy AND
			AzimuthElevationControl.AzimuthAxis.Busy AND
			DerotatorControl.DerotatorAxis.Busy THEN
				Stage := 50;
		END_IF
	50:
		IF NOT ElevationControl.ElevationAxis.Busy AND ElevationControl.ElevationAxis.MoveDone THEN
			ElevationControl.MoveAxis := FALSE;
		END_IF
		IF NOT AzimuthElevationControl.AzimuthAxis.Busy AND AzimuthElevationControl.AzimuthAxis.MoveDone THEN
			AzimuthElevationControl.MoveAxis := FALSE;
		END_IF
		IF NOT DerotatorControl.DerotatorAxis.Busy AND DerotatorControl.DerotatorAxis.MoveDone THEN
			DerotatorControl.MoveAxis := FALSE;
		END_IF
		IF NOT ElevationControl.MoveAxis AND 
           NOT AzimuthElevationControl.MoveAxis AND 
		   NOT DerotatorControl.MoveAxis THEN
		   Stage := 75;
		END_IF
	75:
		IF NOT sliding AND stopped THEN // all axis standstill
			Stage := 100;
		END_IF
	100:
		ElevationControl.MoveAxis := FALSE;
		AzimuthElevationControl.MoveAxis := FALSE;
		DerotatorControl.MoveAxis := FALSE;
		azimuth := azimuth_calc;
		elevation := elevation_calc;
		goto := FALSE;
		// enable automatic tracking
		track := autotrack;
		Stage := 0;
END_CASE
GoToEvent(Trigger := Stage > LastStage, FormatString := 'GoTo progress: %s', OnMessage := USINT_TO_STRING(Stage));
LastStage := Stage;
END_METHOD

METHOD hometelescope : BOOL
VAR_INPUT
END_VAR

VAR
	HomeEvent: FB_Eventlog;
	command_timeout: TON;
END_VAR
command_timeout(IN := NOT hometelescope, PT := T#600S);
IF command_timeout.Q THEN
	error := TRUE;
	errorid := 16#30;
	hometelescope :=TRUE;
END_IF

IF ready AND stopped AND NOT busy AND NOT tracking THEN
	ElevationControl.velocity := 10.0;
	ElevationControl.position := elevation_home;
	ElevationControl.MoveAxis := TRUE;
	AzimuthElevationControl.velocity := 10.0;
	AzimuthElevationControl.position := azimuth_home;
	AzimuthElevationControl.MoveAxis := TRUE;
	DerotatorControl.Velocity := 10.0;
	DerotatorControl.position := 180.0;
	DerotatorControl.MoveAxis := TRUE;	
END_IF

IF ElevationControl.ElevationAxis.MoveDone AND 
	AzimuthElevationControl.AzimuthAxis.MoveDone AND 
	DerotatorControl.DerotatorAxis.MoveDone THEN
	gohome := FALSE;
	elevation := elevation_current;
	azimuth := azimuth_current;
	hometelescope := TRUE;
ELSE
	hometelescope := FALSE;
END_IF

HomeEvent(Trigger := hometelescope, 
			Level := ADSLOG_MSGTYPE_HINT,
			FormatString := '%s',
			OnMessage := 'Telescope is homed.');
END_METHOD

METHOD parktelescope: USINT
VAR_INPUT
END_VAR
VAR
	ParkEvent:	FB_Eventlog;
END_VAR
VAR_STAT
	Stage:		USINT := 0;
	LastStage:	USINT := 101;
END_VAR
parktelescope := Stage;
IF reset OR error THEN
	Stage := 0;
END_IF
IF isparked THEN
	Stage := 100;
END_IF
CASE Stage OF
	0: 
		gohome := 	FALSE;
		track := 	FALSE;
		goto := 	FALSE;
		slew := 	FALSE;
		Focuscontrol.position := 53.6;
		// disable filterwheel
		FilterWheelControl.Enable := FALSE;
		IF Error THEN // emergency park
			HydraulicsControl.close_brake();
			ElevationControl.enable := FALSE;
			AzimuthElevationControl.Enable := FALSE;
			DerotatorControl.enable := FALSE;	
			CoverControl.close := TRUE;	
			Stage := 80;
		END_IF
		Stage := 20;
	20:
		ElevationControl.position := elevation_park;
		ElevationControl.velocity := 10.0;
		ElevationControl.MoveAxis := TRUE;
		AzimuthElevationControl.position := azimuth_park;
		AzimuthElevationControl.velocity := 10;
		AzimuthElevationControl.MoveAxis := TRUE;
		DerotatorControl.position := derotator_park;
		DerotatorControl.Velocity := 10.0;
		DerotatorControl.MoveAxis := TRUE;
		IF ElevationControl.ElevationAxis.Busy AND
			AzimuthElevationControl.AzimuthAxis.Busy AND
			DerotatorControl.DerotatorAxis.Busy THEN
				Stage := 40;
		END_IF
	40:
		IF ElevationControl.ElevationAxis.MoveDone THEN
			ElevationControl.MoveAxis := FALSE;
		END_IF
		IF AzimuthElevationControl.AzimuthAxis.MoveDone THEN
			AzimuthElevationControl.MoveAxis := FALSE;
		END_IF
		IF DerotatorControl.DerotatorAxis.MoveDone THEN
			DerotatorControl.MoveAxis := FALSE;
		END_IF
		IF NOT sliding THEN // all axis standstill
			Stage := 60;
		END_IF
	60:
		IF NOT ElevationControl.enable AND NOT AzimuthElevationControl.Enable AND NOT DerotatorControl.enable THEN
			stage := 80;
		END_IF
		
		IF stopped THEN 
			ElevationControl.enable := FALSE;
			AzimuthElevationControl.Enable := FALSE;
			DerotatorControl.enable := FALSE;
		END_IF
		
		ElevationControl.MoveAxis := FALSE;
		AzimuthElevationControl.MoveAxis := FALSE;
		DerotatorControl.MoveAxis := FALSE;
	80:
		IF ElevationControl.enable OR AzimuthElevationControl.Enable OR DerotatorControl.enable THEN
			stage := 60;
		END_IF
		IF HydraulicsControl.brake_closed THEN
			CoverControl.close := TRUE;
			HydraulicsControl.enable := FALSE;			
		END_IF
		IF CoverControl.isclosed THEN
			Stage := 100;
		END_IF
	100:
			isparked := TRUE;
			park := FALSE;
			parktelescope := 100;
			Stage := 0;	
END_CASE
ParkEvent(Trigger := Stage > LastStage, FormatString := 'Parking progress: %s', OnMessage := USINT_TO_STRING(Stage));
LastStage := Stage;
END_METHOD

METHOD poweron : BOOL
VAR_INPUT
END_VAR
VAR
END_VAR
IF NOT Main.brake_clearing THEN
	powerfailure := TRUE;
	TCSpowerEvent.OnMessage := 'failure: brake clearing not set';
	power := FALSE;
ELSIF NOT Transformer.power_OK THEN
	powerfailure := TRUE;
	TCSpowerEvent.OnMessage := 'failure: main power failure';
	power := FALSE;
ELSIF NOT Transformer.phase_available THEN
	powerfailure := TRUE;
	TCSpowerEvent.OnMessage := 'failure: hydraulics power failure';
	power := FALSE;
ELSIF error THEN
	powerfailure := TRUE;
	TCSpowerEvent.OnMessage := 'Generic error during power on occured.';
	power := FALSE;
ELSE
	powerfailure := FALSE;		
END_IF
// COVER MUST BE OPENED FOR A SUCCESSFUL WAKE & SHAKE COMMAND!
Covercontrol.open := TRUE;

// enable elevation, enable azimuth
IF MAIN.ready AND CoverControl.isopen THEN
	ElevationControl.enable := TRUE;
	AzimuthElevationControl.enable := TRUE;
	DerotatorControl.enable := TRUE;
	FilterWheelControl.Enable := TRUE;
END_IF

IF ElevationControl.Ready AND NOT ElevationControl.Calibrated THEN
	ElevationControl.HomeAxis := TRUE;
END_IF

IF AzimuthElevationControl.ready AND NOT AzimuthElevationControl.calibrated THEN
	AzimuthElevationControl.HomeAxis := TRUE;
END_IF

// enable derotator
IF ElevationControl.Ready THEN
	DerotatorControl.HomeAxis := DerotatorControl.Ready AND NOT DerotatorControl.Calibrated;
END_IF

// home filterwheel after Derotator Axis to avoid additional torque
IF DerotatorControl.Calibrated THEN
	FilterWheelControl.HomeAxis := FilterWheelControl.Ready AND NOT FilterWheelControl.Calibrated;
END_IF

// start calibration of focus after elevation has been calibrated
// this avoids imbalance by the M2 mirror on the elvation during its calibration
IF ElevationControl.Calibrated AND NOT FocusControl.Calibrated THEN
	FocusControl.enable := TRUE;
	FocusControl.HomeAxis := TRUE;
END_IF

IF CoverControl.isopen AND 
	ElevationControl.Calibrated AND
	AzimuthElevationControl.calibrated AND
	DerotatorControl.Calibrated AND
	FilterWheelControl.Calibrated AND
	FocusControl.Calibrated THEN
	power := FALSE;
	poweron := TRUE;
	isparked := FALSE;
	// rest filterwheel until reactivation on filter change
	FilterWheelControl.Enable := FALSE;
	// slew the telescope to the home position
	gohome := TRUE;
ELSE
	poweron := FALSE;
END_IF
END_METHOD

METHOD slewtelescope : USINT
VAR_INPUT
END_VAR
VAR
	SlewEvent:	FB_Eventlog;
	command_timeout: TON;
END_VAR
VAR_STAT
	Stage:		USINT := 0;
	LastStage:	USINT := 101;
END_VAR
slewtelescope := Stage;
command_timeout(IN := Stage < 100, PT := T#600S);
IF command_timeout.Q THEN
	error := TRUE;
	errorid := 16#40;
	slew := FALSE;
	Stage := 0;
END_IF
IF reset OR error THEN
	Stage := 0;
END_IF
CASE Stage OF
	0:	
		IF ready AND stopped AND NOT busy AND NOT tracking THEN
			Stage := 25;
		END_IF
	25:
		ElevationControl.position := elevation;
		ElevationControl.velocity := 10.0;
		ElevationControl.MoveAxis := TRUE;
		AzimuthElevationControl.position := azimuth;
		AzimuthElevationControl.velocity := 10.0;
		AzimuthElevationControl.MoveAxis := TRUE;
		DerotatorControl.position := elevation + derotator_offset;
		DerotatorControl.Velocity := 10.0;
		DerotatorControl.MoveAxis := TRUE;
		IF ElevationControl.ElevationAxis.Busy AND
			AzimuthElevationControl.AzimuthAxis.Busy AND
			DerotatorControl.DerotatorAxis.Busy THEN
				Stage := 50;
		END_IF
	50:
		IF ElevationControl.ElevationAxis.MoveDone THEN
			ElevationControl.MoveAxis := FALSE;
		END_IF
		
		IF AzimuthElevationControl.AzimuthAxis.MoveDone THEN
			AzimuthElevationControl.MoveAxis := FALSE;
		END_IF

		IF DerotatorControl.DerotatorAxis.MoveDone THEN
			DerotatorControl.MoveAxis := FALSE;
		END_IF
		IF NOT sliding AND stopped THEN // all axis standstill
			Stage := 100;
		END_IF
	100:
		ElevationControl.MoveAxis := FALSE;
		AzimuthElevationControl.MoveAxis := FALSE;
		DerotatorControl.MoveAxis := FALSE;
		rightascension := rightascension_calc;
		declination := declination_calc;
		slew := FALSE;
		Stage := 0;
END_CASE
SlewEvent(Trigger := Stage > LastStage, FormatString := 'Slew progress: %s', OnMessage := USINT_TO_STRING(Stage));
LastStage := Stage;
END_METHOD

METHOD stoptelescope : BOOL
VAR_INPUT
END_VAR
ElevationControl.StopAxis := TRUE;
AzimuthElevationControl.StopAxis := TRUE;
DerotatorControl.StopAxis := TRUE;
IF stopped THEN
	ElevationControl.StopAxis := FALSE;
	AzimuthElevationControl.StopAxis := FALSE;
	DerotatorControl.StopAxis := FALSE;
	stop := FALSE;
END_IF
END_METHOD

METHOD tracktelescope : BOOL
VAR_INPUT
END_VAR
// Elevation
DerotatorVelocity := F_Derotatorvelocity(elevation_calc, azimuth_calc, latitude);
ElevationVelocity := F_Elevationvelocity(azimuth_calc, latitude);
AzimuthVelocity := F_Azimuthvelocity(elevation_calc, azimuth_calc, latitude);
IF elevation_current < 5.0 OR elevation_current > 89.5 THEN 
	track := FALSE;
END_IF
IF azimuth_current > 440.0 THEN
	track := FALSE;
END_IF
IF (derotator_current < -69.0 AND DerotatorVelocity<0.0) OR (derotator_current > 379.0 AND DerotatorVelocity>0.0) THEN
	track := FALSE;
END_IF

ElevationControl.position := elevation_calc;
IF NOT ElevationControl.Tracking THEN
	ElevationControl.velocity := 10.0;
	ElevationControl.MoveAxis := TRUE;
	IF NOT ElevationControl.ElevationAxis.Busy AND ElevationControl.ElevationAxis.MoveDone THEN
		ElevationControl.MoveAxis := FALSE;
		IF ElevationControl.ElevationAxis.isTracking THEN
			ElevationControl.velocity := ElevationVelocity;
		ELSE
			ElevationControl.velocity := 3.0*ElevationVelocity;
		END_IF
		ElevationControl.velocity := ElevationVelocity;
		ElevationControl.Tracking := TRUE;
	END_IF
ELSE
	ElevationControl.velocity := ElevationVelocity;
END_IF

// Azimuth
AzimuthElevationControl.position := azimuth_calc;
IF NOT AzimuthElevationControl.Tracking THEN
	AzimuthElevationControl.velocity := 10.0;
	AzimuthElevationControl.MoveAxis := TRUE;
	IF NOT AzimuthElevationControl.AzimuthAxis.Busy AND AzimuthElevationControl.AzimuthAxis.MoveDone THEN
		AzimuthElevationControl.MoveAxis := FALSE;
		IF AzimuthElevationControl.AzimuthAxis.isTracking THEN
			AzimuthElevationControl.velocity := AzimuthVelocity;
		ELSE
			AzimuthElevationControl.velocity := 3.0*AzimuthVelocity;
		END_IF
		AzimuthElevationControl.velocity := AzimuthVelocity;
		AzimuthElevationControl.Tracking := TRUE;
	END_IF
ELSE
	AzimuthElevationControl.velocity := AzimuthVelocity;
END_IF

// Derotator
DerotatorControl.position := derotation_calc;
IF NOT DerotatorControl.Tracking THEN
	DerotatorControl.Velocity := 10.0;
	DerotatorControl.MoveAxis := TRUE;
	IF NOT DerotatorControl.DerotatorAxis.Busy AND DerotatorControl.DerotatorAxis.MoveDone THEN
		DerotatorControl.MoveAxis := FALSE;
		IF DerotatorControl.DerotatorAxis.isTracking THEN
			DerotatorControl.Velocity := DerotatorVelocity;
		ELSE
			DerotatorControl.Velocity := 3.0*DerotatorVelocity;
		END_IF
		DerotatorControl.Velocity := DerotatorVelocity;
		DerotatorControl.Tracking := TRUE;
	END_IF
ELSE
	DerotatorControl.Velocity := DerotatorVelocity;
END_IF
END_METHOD

END_PROGRAM

// ---- POUs/FunctionBlocks/FB_EQ2HOR2.TcPOU
FUNCTION_BLOCK FB_EQ2HOR2
VAR_INPUT
	// right ascension in degrees
	alpha: LREAL;
	// declination in degrees
	delta: LREAL;
	// longitude in degrees
	lon: LREAL;
	// latitude in degrees
	lat: LREAL;
	// Julian Days
	JD: LREAL;
END_VAR
VAR_OUTPUT
	// altitude in degrees
	alt: LREAL;
	// azimuth in degrees
	az: LREAL;
	// hour angle in degreesss
	ha: LREAL;
END_VAR
VAR
	lst: LREAL;
	// helper variables
	sinalt,
	// in radians
	phi_r, tau_r, alpha_r, delta_r: LREAL;
	// current epoch
	J_now: 		LREAL;
	// enable precession
	precess: 	BOOL := TRUE;
	// enable refraction correction
	refract:	BOOL := TRUE;
	// precession function block
	fbprecess: 	FB_PRECESS3;
	//precessed coordinates
	alpha1, delta1:	LREAL;
END_VAR
VAR CONSTANT
	d2r:	LREAL := PI/180.0;
	r2d:	LREAL := 180.0/PI;
END_VAR

(* 
source: http://star-www.st-and.ac.uk/~fv/webnotes/chapter7.htm
https://squarewidget.com/astronomical-calculations-sidereal-time/

*)
lst := ct2lst(lon, jd) * 15.0; // lst in degrees

J_now := (JD - 2451545.0)/365.25 + 2000.0; // compute current equinox
IF precess THEN
	fbprecess( ra := alpha, dec := delta, 
	//EQUINOX1 := 2000.0, EQUINOX2 := J_now, 
	ra_precessed =>alpha1, dec_precessed => delta1);
ELSE
	alpha1 := alpha;
	delta1 := delta;	
END_IF

ha := MODABS(lst - alpha1, 360.0);

alpha_r := alpha1 * d2r;
delta_r := delta1 * d2r;
tau_r := lst*d2r - alpha_r;
phi_r := lat*d2r;

sinalt := SIN(phi_r)*SIN(delta_r) + COS(phi_r)*COS(delta_r)*COS(tau_r);
alt := ASIN(sinalt) * r2d;
IF refract THEN
	alt := alt + Refraction(alt, pressure := 770.0, temperature := 10.0);
END_IF
az := ATAN2(SIN(tau_r), SIN(phi_r)*COS(tau_r) - COS(phi_r)*TAN(delta_r)) * r2d + 180.0;

END_FUNCTION_BLOCK

// ---- POUs/FunctionBlocks/FB_PRECESS3.TcPOU
FUNCTION_BLOCK FB_PRECESS3
VAR_INPUT
	// right ascension in degrees
	ra: LREAL;
	// declination in degrees
	dec: LREAL;
	
END_VAR
VAR_OUTPUT
	// precessed right ascension
	ra_precessed:	LREAL;
	// precessed declination
	dec_precessed:	LREAL;
END_VAR
VAR
	ra_rad, dec_rad: LREAL;
	// starting jd (J2000)
	jd0: LREAL;
	// traget JD
	jd: LREAL;
	t, 
	eta, 
	z, 
	phi,
	A,
	B,
	C	: LREAL;
END_VAR
VAR CONSTANT
	deg_to_rad : LREAL := PI/180.0;
	sec_to_rad : LREAL := deg_to_rad/3600.0;
END_VAR

// see Jean Meeus p.130

ra_rad := ra*deg_to_rad;
dec_rad := dec*deg_to_rad;

// todo epoch to jd and jd0
JD := TelescopeControl.jd;
jd0 := 2451545.0;
t := (jd - jd0) / 36525.0;

eta :=	(2306.2181*t + 0.30188*t*t + 0.017998*t*t*t) * sec_to_rad;
z :=	(2306.2181*t + 1.09468*t*t + 0.018203*t*t*t) * sec_to_rad;
phi :=	(2004.3109*t - 0.42665*t*t - 0.041833*t*t*t) * sec_to_rad;

A :=            COS(dec_rad) * SIN(ra_rad + eta);
B := COS(phi) * COS(dec_rad) * COS(ra_rad + eta) - SIN(phi) * SIN(dec_rad);
C := SIN(phi) * COS(dec_rad) * COS(ra_rad + eta) + COS(phi) * SIN(dec_rad);

// tan(ra - z) == A/B
ra_precessed := MODABS((ATAN2(A, B) + z)/deg_to_rad, 360);
IF ABS(dec) > 89.5 THEN
	dec_precessed := ACOS(SQRT(A*A + B*B))/deg_to_rad;
ELSE
	// sin(de)c = C
	dec_precessed := ASIN(C)/deg_to_rad;	
END_IF

END_FUNCTION_BLOCK

// ---- POUs/Functions/ATAN2.TcPOU
FUNCTION ATAN2 : LREAL
VAR_INPUT
	y, x: LREAL;
END_VAR
VAR
END_VAR

(* source: https://de.wikipedia.org/wiki/Arctan2 *)
ATAN2 := 0.0;

IF x > 0 THEN
	ATAN2 := ATAN(y/x);
ELSIF x < 0 AND y > 0 THEN
	ATAN2 := ATAN(y/x) + PI;
ELSIF x < 0 AND y = 0 THEN
	ATAN2 := PI;
ELSIF x < 0 AND y < 0 THEN
	ATAN2 := ATAN(y/x) - PI;
ELSIF x = 0 AND y > 0 THEN
	ATAN2 := PI/2.0;
ELSIF x = 0 AND y < 0 THEN
	ATAN2 := -PI/2.0;
END_IF

END_FUNCTION

// ---- POUs/Functions/Refraction.TcPOU
FUNCTION Refraction : LREAL
VAR_INPUT
	// elevation in degrees
	elevation: LREAL;
	// pressure in mBar
	pressure: LREAL := 770.0;
	// temperature in Celsius
	temperature : LREAL := 10.0;
END_VAR
VAR
END_VAR
VAR CONSTANT
	d2r:	LREAL := PI/180.0;
END_VAR

// sanity checks
elevation := LIMIT(0.0, elevation, 90.0);
pressure := LIMIT(600.0, pressure, 1200.0);
temperature := LIMIT(-30.0, temperature, 40.0);
// refraction in arcmin
Refraction := 1.02 / TAN((elevation + 10.3/(elevation + 5.11)) * d2r);
Refraction := Refraction * pressure * 283.0 / (1010.0 * (273.0 * temperature));
//refraction in degrees
Refraction := Refraction / 60.0;

END_FUNCTION

// ---- POUs/FunctionBlocks/FB_HOR2EQ.TcPOU
FUNCTION_BLOCK FB_HOR2EQ
VAR_INPUT
	//altitude (in degrees) [scalar OR vector]
	alt: LREAL;  
	//azimuth angle (in degrees, measured EAST from NORTH, but see keyword WS below.) [scalar or vector]
	az: LREAL;
	// Julian Date [scalar or vector], double precision
	JD: 		LREAL;
	lat:		LREAL;
	lon:		LREAL;
	WS:			BOOL;
	precess:	BOOL := FALSE;
	NUTATE:		BOOL := FALSE;
	aberration:	BOOL := FALSE;
	refract:	BOOL := FALSE;
	altitude:	LREAL := 0.0;
END_VAR
VAR_OUTPUT
	// Right Ascension of object  (J2000) in degrees (FK5)
	ra: 	LREAL;
	// Declination of object (J2000) in degrees (FK5)
	dec:	LREAL;
	// hour angle (in degrees) (optional)
	ha:		LREAL;
END_VAR
VAR
	
	alt_,
	az_,
	lmst,
	J_now: LREAL;
	co_nutate: 		FB_CO_NUTATE;
	co_aberration: 	CO_ABERRATION;
	co_refract:		CO_REFRACT;
	fbprecess:		FB_PRECESS;
	altaz2hadec:	FB_ALTAZ2HADEC;
	last: LREAL;
	dra1: LREAL;
	ddec1: LREAL;
	eps: LREAL;
	d_psi: LREAL;
	dra2: LREAL;
	ddec2: LREAL;
END_VAR
VAR CONSTANT
	//d2r:	LREAL := PI/180.0;
	//r2d:	LREAL := 180.0/PI;
	//h2r:	LREAL := PI/12.0;
	h2d:	LREAL := 15.0;
END_VAR



alt_ := alt;   //do this so we don't change ra, dec arrays.
az_ := az;


//*******************************************************************************************
// Make Correction for ATMOSPHERIC REFRACTION
// (use this for visible and radio wavelengths; author is unsure about other wavelengths)
IF refract THEN 
	co_refract(	old_alt := alt, 
				altitude := altitude, 
				to_observed := TRUE, 
				new_alt => alt);
END_IF

IF WS THEN 
	az_ := az_ - 180.0;
END_IF

co_nutate(	jd := jd, 
			ra := 45.0, 
			dec := 45.0, 
			d_ra => dra1, 
			d_dec => ddec1, 
			eps => eps, 
			d_psi => d_psi);
//******************************************************************************
//Calculate LOCAL APPARENT SIDEREAL TIME
// first get local mean sidereal time (lmst)
// get LST (in hours) - note:this is indep of tzone since giving jd
lmst := ct2lst( lon, jd);
// convert LMST TO degrees (btw, THIS is the RA OF the zenith)
lmst := lmst*h2d;
// calculate local APPARENT sidereal time (last)
// ADD correction in degrees
last := lmst + d_psi *COS(eps)/3600.0 ; 

//****************************************************************************
// Now do the spherical trig to get APPARENT Hour Angle [degrees], and
// declination [degrees].
altaz2hadec( alt := alt_, az := az_, lat := lat, ha => ha, dec => dec);

// Find Right Ascension (in degrees, from 0 to 360.)
 ra := MODABS(last - ha + 360.0, 360.0);



//*****************************************************************************
// calculate NUTATION and ABERRATION Corrections to Ra-Dec
IF NUTATE THEN
	co_nutate(	jd := jd, 
			ra := ra, 
			dec := dec, 
			d_ra => dra1, 
			d_dec => ddec1, 
			eps => eps, 
			d_psi => d_psi);
ELSE
	dra1 := 0.0;
	ddec1 := 0.0;	
END_IF
IF aberration THEN
	co_aberration(	jd := jd, 
				ra := ra, 
				dec := dec, 
				d_ra => dra2, 
				d_dec => ddec2, 
				eps := eps);
ELSE
	dra2 := 0.0;
	ddec2 := 0.0;	
END_IF
//******************************************************************************
// Make Nutation and Aberration Corrections (if wanted)

ra := ra - (dra1 + dra2)/3600.0;
dec := dec - (ddec1 + ddec2)/3600.0;
 //compute current equinox
J_now := (JD - 2451545.0)/365.25 + 2000.0 ;

//*****************************************************************************
// PRECESS coordinates to current date
// (uses astro lib procedure PRECESS.pro)

IF precess THEN 
	fbprecess( ra := ra, dec := dec, 
	EQUINOX1 := 2000.0, EQUINOX2 := J_now, 
	ra_precessed =>ra, dec_precessed => dec);                   
END_IF

END_FUNCTION_BLOCK

// ---- POUs/FunctionBlocks/FB_CO_NUTATE.TcPOU
FUNCTION_BLOCK FB_CO_NUTATE
VAR_INPUT
	jd,
	ra,
	dec:	LREAL;
END_VAR
VAR_OUTPUT
	d_ra,
	d_dec,
	eps,
	d_psi,
	d_eps:	LREAL;
END_VAR
VAR
	T, 
	eps0,
ce, se,x,y,z,x2,y2,z2,rad,xyproj,ra2,dec2: LREAL;
	nutate:	FB_NUTATE;
END_VAR
VAR CONSTANT
	d2r:	LREAL := PI/180.0;
	d2as:	LREAL := PI/(180.0*3600.0);
END_VAR

// Julian centuries FROM J2000 OF jd.
T := (jd -2451545.0)/36525.0; 

// must calculate obliquity OF ecliptic
nutate(jd := jd,
		nut_long => d_psi, 
		nut_obliq => d_eps); 

eps0 := 23.4392911*3600.0 - 46.8150*T - 0.00059*EXPT(T, 2) + 0.001813*EXPT(T, 3);
eps := (eps0 + d_eps)/3600.0*d2r; // TRUE obliquity OF the ecliptic in radians
 
//useful numbers
ce := COS(eps);
se := SIN(eps);

// convert ra-dec to equatorial rectangular coordinates
x := COS(ra*d2r) * COS(dec*d2r);
y := SIN(ra*d2r) * COS(dec*d2r);
z := SIN(dec*d2r);

// apply corrections to each rectangular coordinate
x2 := x - (y*ce + z*se)*d_psi * d2as;
y2 := y + (x*ce*d_psi - z*d_eps) * d2as;
z2 := z + (x*se*d_psi + y*d_eps) * d2as;

// convert back to equatorial spherical coordinates
rad := SQRT(x2*x2 + y2*y2 + z2*z2);
xyproj := SQRT(x2*x2 + y2*y2);

ra2  := x2 * 0.0;
dec2 := x2 * 0.0;

// Calculate Ra and Dec in RADIANS (later convert to DEGREES)
IF (xyproj = 0) AND (z <> 0) THEN
	// places where xyproj=0 (point at NCP or SCP)
	dec2 := ASIN(z2/rad);
	ra2 := 0.0;
END_IF
 
IF (xyproj <> 0) THEN
	// places other than NCP or SCP
	ra2 := ATAN2(y2, x2);
	dec2 := ASIN(z2/rad);
END_IF

// convert to DEGREES

ra2 := ra2 /d2r;
dec2 := dec2 /d2r;

ra2 := MODABS(ra2, 360.0);


// Return changes in ra and dec in arcseconds
d_ra := (ra2 - ra) * 3600.0;
d_dec := (dec2 - dec) * 3600.0;

END_FUNCTION_BLOCK

// ---- POUs/FunctionBlocks/CO_REFRACT.TcPOU
FUNCTION_BLOCK CO_REFRACT
VAR_INPUT
	old_alt: LREAL;
	altitude: LREAL := 0.0;
	pressure: LREAL := 0.0;
	temperature: LREAL := 0.0;
	epsilon: LREAL := 0.25; //accuracy of iteration for observed=TRUE case, in arcseconds
	TO_OBSERVED: BOOL;
END_VAR
VAR_OUTPUT
	new_alt: LREAL;
END_VAR
VAR
	aout, P, T, dr, cur, last : LREAL;
END_VAR
VAR CONSTANT
	alpha : LREAL := 0.0065; //temp lapse rate [deg C per meter]
END_VAR

IF temperature = 0.0 THEN
	IF altitude > 11000.0 THEN 
		temperature := 211.5; 
	ELSE 
		temperature := 283.0 - alpha*altitude;
	END_IF
END_IF

// estimate Pressure based on altitude, using U.S. Standard Atmosphere formula.
IF pressure = 0 THEN 
	pressure := 1010.0*EXPT(1-6.5/288000*altitude, 5.255);
END_IF

IF NOT TO_OBSERVED THEN 
	aout := old_alt - co_refract_forward(old_alt, P:=pressure,T:=temperature);
ELSE
	aout := 0.0;
	P := pressure; T := temperature;
	//calculate initial refraction guess
	dr := co_refract_forward(old_alt, P:=P, T:=T);
	cur := old_alt + dr; // guess of observed location

	REPEAT 
	 	last := cur;
		dr := co_refract_forward(cur, P:= P, T:=T);
	  	cur := old_alt + dr;
	UNTIL ABS(last-cur)*3600.0 < epsilon
	END_REPEAT
	aout := cur;
END_IF

new_alt := aout;

END_FUNCTION_BLOCK

// ---- POUs/FunctionBlocks/FB_PRECESS.TcPOU
FUNCTION_BLOCK FB_PRECESS
VAR_INPUT
	ra, 
	dec,
	equinox1,
	equinox2: LREAL;
	RADIAN:	BOOL := FALSE;
END_VAR
VAR_OUTPUT
	ra_precessed,
	dec_precessed:	LREAL;
END_VAR
VAR
	ra_rad, dec_rad: LREAL;
	a,b,c,t: LREAL;
	x, x2: ARRAY[0..2] OF LREAL;
	st1: LREAL;
	rot: ARRAY[0..2,0..2] OF LREAL;
	sina, sinb, sinc, cosa,cosb,cosc: LREAL;
END_VAR
VAR CONSTANT
	deg_to_rad : LREAL := PI/180.0;
	sec_to_rad : LREAL := deg_to_rad/3600.0;
END_VAR

IF NOT RADIAN THEN
	ra_rad := ra*deg_to_rad;
	dec_rad := dec*deg_to_rad;
ELSE
    //Convert TO double precision IF NOT already
	ra_rad := ra;
	dec_rad := dec;
END_IF

a := COS( dec_rad );
x[0] := a*COS(ra_rad); x[1] := a*SIN(ra_rad); x[2] := SIN(dec_rad);

//*** PREMAT code starts here
ST1 := 0.001*( equinox1 - 2000.0);
t := 0.001*( equinox2 - equinox1);
//  Compute 3 rotation angles
A := sec_to_rad * T * (23062.181 + ST1*(139.656 +0.0139*ST1) + T*(30.188 - 0.344*ST1+17.998*T));
B := sec_to_rad * T * T * (79.280 + 0.410*ST1 + 0.205*T) + A;
C := sec_to_rad * T * (20043.109 - ST1*(85.33 + 0.217*ST1) + T*(-42.665 - 0.217*ST1 -41.833*T));
  sina := SIN(a); sinb := SIN(b);  sinc := SIN(c);
  cosa := COS(a); cosb := COS(b);  cosc := COS(c);

rot[0,0] :=  cosa*cosb*cosc-sina*sinb; 	rot[0,1] := sina*cosb+cosa*sinb*cosc; 	rot[0,2] := cosa*sinc;
rot[1,0] := -cosa*sinb-sina*cosb*cosc; 	rot[1,1] := cosa*cosb-sina*sinb*cosc; 	rot[1,2] := -sina*sinc;
rot[2,0] := -cosb*sinc;					rot[2,1] := -sinb*sinc; 				rot[2,2] := cosc;

//*** PREMAT code ends here

//x2 := rot* x; //rotate to get output direction cosines
x2[0] := rot[0,0]*x[0] + rot[1,0]*x[1] + rot[2,0]*x[2];
x2[1] := rot[0,1]*x[0] + rot[1,1]*x[1] + rot[2,1]*x[2];
x2[2] := rot[0,2]*x[0] + rot[1,2]*x[1] + rot[2,2]*x[2];

ra_rad := atan2(x2[1],x2[0]);
dec_rad := ASIN(x2[2]);

IF NOT RADIAN THEN
	ra_precessed := ra_rad/deg_to_rad;
	ra_precessed := MODABS(ra_precessed, 360.0);            //RA between 0 AND 360 degrees
	dec_precessed := dec_rad/deg_to_rad;
ELSE
	ra_precessed := ra_rad; 
	dec_precessed := dec_rad;
	ra_precessed := MODABS(ra_rad, 2.0*PI);
END_IF

END_FUNCTION_BLOCK

// ---- POUs/TelescopeAuxiliary.TcPOU
PROGRAM TelescopeAuxiliary
VAR
	MQTTTimer : TON := (PT:=T#5S);
	cycle:	USINT;
	FBReadPressure : FB_ReadAdsSymByName;
	FBReadTemperature: FB_ReadAdsSymByName;
	// EL3064-1
	raw_dewar_pressure		AT%I*: INT;
	pressure_voltage:	REAL;
	dewar_warning_trigger: SR;
	dewar_error_trigger: SR;
	DewarWarning, DewarError: FB_EventLog;
END_VAR
VAR_OUTPUT
	// BT9 mirror
	temperature_mirror2:	REAL;
	// BT10
	temperature_mirror1:	REAL;
	pressure:		REAL;
	temperature:	REAL;
	dewar_pressure:	REAL;
	dewar_pressure_atm: REAL;
END_VAR

temperature_mirror1 := GVL_Telescope.temperature_mirror1 / 1000.0;
temperature_mirror2 := GVL_Telescope.temperature_mirror2 / 1000.0;


cycle := cycle MOD 8;
FBReadPressure(
	bRead := cycle MOD 10 = 1,
	sNetId := '5.40.71.146.1.1',
	sVarName := 'Environment.Pressure',
	nDestAddr := ADR(pressure),
	nLen := SIZEOF(pressure),
 	eComMode := eAdsComModeFastCom
	);
FBReadTemperature(
	bRead := cycle MOD 10 = 4,
	sNetId := '5.40.71.146.1.1',
	sVarName := 'Environment.Temperature1',
	nDestAddr := ADR(temperature),
	nLen := SIZEOF(temperature),
 	eComMode := eAdsComModeFastCom
	);
IF NOT (FBReadPressure.bBusy OR FBReadPressure.bError) AND 
   NOT (FBReadTemperature.bBusy OR FBReadTemperature.bError) THEN
	cycle := cycle + 1;
END_IF

pressure_voltage := F_YREAL(raw_dewar_pressure, 0, 32767, 0.0, 10.0);
dewar_pressure := LREAL_TO_REAL(EXPT(10.0, F_YREAL(pressure_voltage, 2.0, 10.0, -9.0, 3.0)));
dewar_pressure_atm := LREAL_TO_REAL(EXPT(10.0, F_YREAL(pressure_voltage, 2.0, 10.0, -7.0, 5.0)));

dewar_warning_trigger(SET1 := dewar_pressure_atm > 1E-6, RESET := dewar_pressure_atm < 5E-7);
dewar_error_trigger(SET1 := dewar_pressure_atm > 1E-5, RESET := dewar_pressure_atm < 1E-6);

DewarWarning(Trigger := dewar_warning_trigger.Q1,
				Level := ADSLOG_MSGTYPE_WARN,
				FormatString := '%s',
				OnMessage := 'Dewar pressure is above nominal.',
				OffMessage := 'Dewar pressure is nominal.');

DewarError(Trigger := dewar_error_trigger.Q1,
				Level := ADSLOG_MSGTYPE_ERROR,
				FormatString := '%s',
				OnMessage := 'Dewar pressure is critical!');


MQTTTimer(IN:=TRUE);
IF MQTTTimer.Q THEN // publish new payload every second

	MAIN.MQTTClient.Publish('telescope', 'dome', 'Mirror1Temperature',	LREAL_TO_FMTSTR(temperature_mirror1, 2, TRUE));
	MAIN.MQTTClient.Publish('telescope', 'dome', 'Mirror2Temperature',	LREAL_TO_FMTSTR(temperature_mirror2, 2, TRUE));
	MAIN.MQTTClient.Publish('telescope', 'dome', 'DewarPressureVoltage', LREAL_TO_FMTSTR(pressure_voltage, 3, TRUE));
	MAIN.MQTTClient.Publish('telescope', 'dome', 'DewarPressure', LREAL_TO_FMTSTR(dewar_pressure_atm, 9, TRUE));
	
	MQTTTimer(IN:=FALSE);

END_IF

END_PROGRAM

// ---- POUs/Functions/DateTime2JD.TcPOU
FUNCTION DateTime2JD : LREAL
VAR_INPUT
	epoch: TIMESTRUCT;
END_VAR
VAR
	a,y,m,d,jdn: LREAL;
END_VAR

(*    import datetime
    from math import floor
    if not type(epoch) is datetime.datetime:
        raise TypeError('datetime must be of type datetime')
    
    a = floor((14 - epoch.month)/12)
    y = epoch.year + 4800 - a
    m = epoch.month + 12*a - 3
    
    d = epoch.day
    d += epoch.hour/24. + epoch.minute/1440. + epoch.second/86400. # microsecond might be added here?
    
    if [epoch.year,epoch.month,d] >= [1582,10,15]:
        jdn = epoch.day + floor((153*m + 2)/5) + 365*y + floor(y/4) - floor(y/100) + floor(y/400) - 32045
    elif [epoch.year,epoch.month,d] <= [1582,10,4]:
        jdn = epoch.day + floor((153*m + 2)/5) + 365*y + floor(y/4) - 32083
    return jdn + (epoch.hour-12)/24. + epoch.minute/1440. + epoch.second/86400.
*)
a := FLOOR((14.0 - epoch.wMonth)/12.0);
y := epoch.wYear + 4800.0 - a;
m := epoch.wMonth + 12.0*a - 3.0;

d := epoch.wDay + (epoch.wHour/24.0) + (epoch.wMinute/1440.0) + (epoch.wSecond/86400.0);

//IF (epoch.wYear > 1582) (* AND (epoch.wMonth > 10.0) AND (d > 15.0)*) THEN
	jdn := epoch.wDay + FLOOR((153*m + 2)/5) + 365.0*y + FLOOR(y/4) - FLOOR(y/100) + FLOOR(y/400) - 32045.0;
//ELSIF (epoch.wYear < 1582) AND (epoch.wMonth < 10) AND (d > 4.0) THEN
//	jdn := epoch.wDay + FLOOR((153*m + 2)/5) + 365.0*y + FLOOR(y/4) - 32083.0;
//END_IF

DateTime2JD := jdn
			+ (epoch.wHour-12.0)/24.0
			+ (epoch.wMinute/1440.0) 
			+ (epoch.wSecond/86400.0)
			+ (DWORD_TO_REAL(epoch.wMilliseconds)/86400000.0);

END_FUNCTION

// ---- POUs/Functions/PointingModelElevation.TcPOU
FUNCTION PointingModelElevation : LREAL
// https://aro.as.arizona.edu/~aro/12_obs_manual/pdfs/Appendix_A_Rev_2.pdf
VAR_INPUT
	// current azimuth of telescope
	azimuth: LREAL;
	// current elevation of telescope
	elevation: LREAL;
	// elevation encoder zero offset
	EOFF: 	LREAL;
	// azimuth axis offset/misalignment north-south
	AN_E:	LREAL;
	// azimuth axis offset/misalignment east-west
	AE_E:	LREAL;
	// gravitational flexure correction at the horizon
	TF:		LREAL;
END_VAR
VAR
END_VAR
VAR CONSTANT
	d2r:	LREAL := PI/180.0;
	//r2d:	LREAL := 180.0/PI;
END_VAR

PointingModelElevation := EOFF + AN_E*COS(azimuth * d2r) + AE_E*SIN(azimuth * d2r) + TF*COS(elevation * d2r);

END_FUNCTION

// ---- POUs/Functions/PointingModelAzimuth.TcPOU
FUNCTION PointingModelAzimuth : LREAL
// https://aro.as.arizona.edu/~aro/12_obs_manual/pdfs/Appendix_A_Rev_2.pdf
VAR_INPUT
	// current azimuth of telescope in degrees
	azimuth: LREAL;
	// current elevation of telescope in degrees
	elevation: LREAL;
	// azimuth encoder zero offset
	AOFF: 	LREAL;
	// collimation error of the electromagnetic axis
	BNP:	LREAL;
	// azimuth axis offset/misalignment north-south
	AN_A:	LREAL;
	// azimuth axis offset/misalignment east-west,
	AE_A:	LREAL;
	// Non-perpendicularity between the mount azimuth and elevation axes
	NPAE:	LREAL;
END_VAR
VAR
	tan_elevation:	LREAL;
	cos_elevation:	LREAL;
END_VAR
VAR CONSTANT
	d2r:	LREAL := PI/180.0;
	//r2d:	LREAL := 180.0/PI;
END_VAR

IF elevation<89.9 THEN
	tan_elevation := TAN(elevation * d2r);
	cos_elevation := COS(elevation * d2r);
ELSE // clamp values so that we do not run into DIV by zero or overflow
	tan_elevation := 572.9572133543033;
	cos_elevation := 0.0017453283658982613;
END_IF

//d(az)=AOFF-BNP/cos(el)+NPAE*tan(el)+AAN*sin(az)*tan(el)-AAE*cos(az)*tan(el)

PointingModelAzimuth := AOFF - BNP/cos_elevation + AN_A*SIN(azimuth * d2r)*tan_elevation - AE_A*COS(azimuth * d2r)*tan_elevation + NPAE*tan_elevation;

END_FUNCTION

// ---- POUs/Functions/F_DerotatorPosition2.TcPOU
FUNCTION F_DerotatorPosition2 : LREAL
VAR_INPUT
	// azimuth of the target
	azimuth: LREAL;
	// elevation of the target in degrees
	elevation: LREAL;
	// declination of the target in degrees
	declination: LREAL;
	// latitude in degrees
	latitude:	LREAL;
	// sign for elevation
	sign:	LREAL := 1.0;
END_VAR
VAR
	// parallactic angle
	de, az, el, la: LREAL;
	parallactic_angle:	LREAL;
	//zenith_distance: LREAL;
END_VAR
VAR CONSTANT
	d2r:	LREAL := PI/180.0;
	r2d:	LREAL := 180.0/PI;
	//h2r:	LREAL := PI/12.0;
	//h2d:	LREAL := 15.0;
END_VAR

// calculate the parallactic angle
de := LIMIT(-90.0, declination, 90.0) * d2r;
az := MODABS(azimuth, 360.0) * d2r;
el := LIMIT(0.0, elevation, 90.0) * d2r;
la := LIMIT(-90.0, latitude, 90.0) * d2r;

parallactic_angle := - r2d * ATAN2(SIN(az), TAN(la)*COS(el)-SIN(el)*COS(az));

F_DerotatorPosition2 := parallactic_angle - sign * elevation;
F_DerotatorPosition2 := MODABS(F_DerotatorPosition2, 360.0);

END_FUNCTION

// ---- POUs/Functions/F_Derotatorvelocity.TcPOU
FUNCTION F_Derotatorvelocity : LREAL
VAR_INPUT
	// elevation in degrees
	elevation: 	LREAL;
	// azimuth in degrees
	azimuth:	LREAL;
	// observers latitude in degrees
	latitude:	LREAL;
END_VAR
VAR
END_VAR
VAR CONSTANT
	// Earth's angular rotation frequency in [deg/s]
	Omega: LREAL := 4.178074605556E-3;
	d2r:	LREAL := PI/180.0;
	//r2d:	LREAL := 180.0/PI;
END_VAR

(* 
source: https://github.com/cytan299/field_derotator/blob/master/field_derotator_formula/field_derotator_formula.pdf
https://circuitcellar.com/research-design-hub/projects/field-derotator-for-astrophotography-part-1/

returns the rotational velocity for the de-rotator in degrees per second
azimuth, latitutde and elevation are converted to radians
*)
IF ABS(COS(elevation * d2r))> 1.0e-3 THEN
	F_Derotatorvelocity := -Omega * COS(azimuth * d2r) * COS(latitude * d2r) / COS(elevation * d2r)  - Omega *COS(latitude * d2r) * SIN(azimuth * d2r);
ELSE
	F_Derotatorvelocity := 0.0;	
END_IF

END_FUNCTION

// ---- POUs/Functions/F_Elevationvelocity.TcPOU
FUNCTION F_Elevationvelocity : LREAL
VAR_INPUT
	// azimuth in degrees
	azimuth:	LREAL;
	// observers latitude in degrees
	latitude:	LREAL;
END_VAR
VAR
END_VAR
VAR CONSTANT
	// Earth's angular rotation frequency in [deg/s]
	Omega: LREAL := 4.178E-3;
	d2r:	LREAL := PI/180.0;
	//r2d:	LREAL := 180.0/PI;
END_VAR

//returns the rotational velocity for the azimuth in degrees per second
F_Elevationvelocity := SIN(azimuth*d2r) * COS(latitude*d2r) * Omega;

END_FUNCTION

// ---- POUs/Functions/F_Azimuthvelocity.TcPOU
FUNCTION F_Azimuthvelocity : LREAL
VAR_INPUT
	// elevation in degrees
	elevation: 	LREAL;
	// azimuth in degrees
	azimuth:	LREAL;
	// observers latitude in degrees
	latitude:	LREAL;
END_VAR
VAR
END_VAR
VAR CONSTANT
	// Earth's angular rotation frequency in [deg/s]
	Omega: LREAL := 4.178E-3;
	d2r:	LREAL := PI/180.0;
	//r2d:	LREAL := 180.0/PI;
END_VAR

IF ABS(COS(elevation * d2r))> 1.0e-3 THEN
	F_Azimuthvelocity := (SIN(latitude * d2r) - COS(latitude * d2r) * COS(azimuth * d2r) * TAN(elevation *d2r))* Omega;
ELSE
	F_Azimuthvelocity := 0.0;	
END_IF

END_FUNCTION

// ---- POUs/SafetyHandling.TcPOU
PROGRAM SafetyHandling
VAR
	// power on delay
	start_delay 	: TON := (PT := T#2S);
	// pulse for error acknowledgement
	ErrAck_Pulse	: TP := (PT := T#500MS);
	// pulse for safety restart
	restart_Pulse 	: TP := (PT := T#500MS);
	// trigger for falling edge of error acknowledgement
	ErrAck_Trigger	: F_TRIG;
	// Errack logging
	ErrAckLog		: FB_EventLog;
	// restart logging
	RestartLog		: FB_EventLog;
	// safety logging
	SafetyLog		: FB_EventLog;
	
END_VAR
VAR_OUTPUT
	// error condition
	Error			: BOOL;
	// Emergency_stop engaged
	Emergency_stop	: BOOL;
END_VAR
VAR_INPUT
	// issue a remote restart
	remote_restart:		BOOL;
	// issue a remote Error Acknowledgment
	remote_ErrAck:		BOOL;
	// issue a remute run/stop
	remote_run:			BOOL := TRUE;
END_VAR

// Safety aus running on start
GVL_Safety.Run := remote_run;
// power on delay for Safety RESTART after RUN=1

// wait n seconds after Start ...
start_delay(IN := Transformer.power_ok);
// ... and send ErrAck for n milliseconds
ErrAck_Pulse(IN := (GVL_Safety.State = 2) AND start_delay.Q);

// Error Acknowledgment: Turn key_switch OFF and press STOP 
GVL_Safety.ErrAck := (NOT GVL_Main.key_switch_remote)
					OR ErrAck_Pulse.Q
					OR remote_ErrAck;
// detect falling edge 
ErrAck_Trigger(CLK := GVL_Safety.ErrAck);
// send restart pulse on falling edge of ErrAck
restart_pulse(IN := ErrAck_Trigger.Q);

// RESTART Safety after pushing reset or power on delay
GVL_Safety.Restart := (Main.reset AND NOT GVL_Main.key_switch_remote) 
					 	OR restart_pulse.Q 
						OR remote_restart;
				
Error := GVL_Safety.Error OR (GVL_Safety.State <> 1);

Emergency_stop := NOT GVL_Safety.Stop;

ErrAckLog(	Trigger := GVL_Safety.ErrAck,
			OnMessage := 'Safety error was acknowledged.');
			
RestartLog(	Trigger := GVL_Safety.Restart,
			Level := ADSLOG_MSGTYPE_WARN,
			OnMessage := 'Safety was restarted.');

SafetyLog(	Trigger := Error,
			Level := ADSLOG_MSGTYPE_ERROR,
			OnMessage := 'Safety Error! Emergency stop enganged!',
			OffMessage := 'Safety is OK.',
			OffLevel := ADSLOG_MSGTYPE_HINT);

END_PROGRAM

// ---- POUs/Transformer.TcPOU
PROGRAM Transformer
VAR_INPUT
	// reset signal for the error condition
	reset_error:		BOOL := FALSE;
	// signal to start the transformer
	softstart_trafo:	BOOL;
END_VAR
VAR_OUTPUT
	// indicates the phases for the hydraulics
	phase_available:	BOOL;
	// trafo failed to start after timeout
	power_failure:		BOOL;
	// restart was inhibited
	restart_inhibited:	BOOL;
END_VAR
VAR
	// watchdog for trafo softstarter
	power_watchdog: 	TON;
	// timer to measure the startup time
	power_timer:		FB_timer;
	// timeout for the startup
	startup_timeout:	TIME := T#5S;
	// error state
	power_error_state:	SR;
	// restart inhibitor
	restart_inhibit:	TOF;
	PowerEvent:			FB_EventLog;
	PowerLog:			FB_EventLog;
	
END_VAR

power_timer(bStart := GVL_Main.softstart_trafo, bStop := power_OK);
power_watchdog(IN := GVL_Main.softstart_trafo AND NOT power_OK,
				PT := startup_timeout,
				Q => power_failure);
power_error_state(SET1 := power_failure, RESET := reset_error);
restart_inhibit(IN := GVL_MAIN.trafo_bypassed, PT := T#5S);

restart_inhibited := NOT GVL_MAIN.trafo_bypassed AND restart_inhibit.Q;
IF restart_inhibited THEN
	softstart_trafo := FALSE;
END_IF
GVL_Main.softstart_trafo := softstart_trafo AND NOT error;

	
phase_available := TRUE; (*GVL_Main.L1L2_voltage > 360.0 AND
					GVL_Main.L2L3_voltage > 360.0 AND
					GVL_Main.L3L1_voltage > 360.0; *)

PowerEvent(	
	Trigger := 		power_failure, 
	Level := 		ADSLOG_MSGTYPE_ERROR,
	FormatString :=	'%s',
	OnMessage := 	'Servo power FAILURE!',
	OffMEssage := 	'Servo power OK');
PowerLog(	
	Trigger := 		power_OK, 
	Level := 		ADSLOG_MSGTYPE_HINT,
	FormatString :=	'%s',
	OnMessage := 	'Mains power is ON',
	OffMEssage := 	'Mains power is OFF');

PROPERTY error : BOOL
GET
error := power_error_state.Q1;
END_GET
END_PROPERTY

PROPERTY power_ok : BOOL
// indicates the power state for the AX5000
GET
power_ok := GVL_main.trafo_bypassed;
END_GET
END_PROPERTY

METHOD reset : BOOL
VAR_INPUT
END_VAR
IF error THEN
	reset_error := TRUE;
ELSE
	reset_error := FALSE;
END_IF
END_METHOD

METHOD start : BOOL
VAR_INPUT
END_VAR
softstart_trafo := TRUE;
END_METHOD

PROPERTY startup_time : TIME
GET
startup_time := power_timer.tDifference;
END_GET
SET
startup_timeout := startup_time;
END_SET
END_PROPERTY

METHOD stop : BOOL
VAR_INPUT
END_VAR
softstart_trafo := FALSE;
END_METHOD

END_PROGRAM

// ---- POUs/FunctionBlocks/FB_EQ2HOR.TcPOU
FUNCTION_BLOCK FB_EQ2HOR
VAR_INPUT
	RA: 		LREAL;	// Right Ascension of object  (J2000) in degrees (FK5)
	Dec: 		LREAL;	// Declination of object (J2000) in degrees (FK5)
	JD: 		LREAL;	// Julian Date
	LAT: 		LREAL;	// north geodetic latitude of location in degrees
	LON: 		LREAL; 	// EAST longitude of location in degrees (Specify west longitude with a negative sign.)
	ALTITUDE:	LREAL := 0.0;  // The altitude of the observing location, in meters. [default=0].  
	WS:			BOOL := FALSE; //  Set this to TRUE get the azimuth measured westward FROM south (NOT East of North).
	PRECESS:	BOOL := TRUE; // Set this to 1 to force precession [default], 0 for no precession correction
	NUTATE:		BOOL := TRUE; // Set this to 1 to force nutation [default], 0 for no nutation.
	ABERRATION:	BOOL := TRUE; // Set this to 1 to force aberration correction [default], 0 for no correction.
	REFRACT:	BOOL := TRUE; // Set to 1 to force refraction correction [default], 0 for no correction.
END_VAR
VAR_OUTPUT
	alt: 	LREAL; // altitude (in degrees)
	az:		LREAL; // azimuth angle (in degrees, measured EAST FROM NORTH, but see keyword WS above.)
	ha:		LREAL; // hour angle (in degrees) (optional)	
END_VAR
VAR
	ra_, dec_, tstart, J_now: LREAL;
	s_now: STRING;
	fbprecess: FB_PRECESS;
	lmst: LREAL;
	last: LREAL;
	d_psi: LREAL;
	eps: LREAL;
	hadec2altaz:	FB_HADEC2ALTAZ;
	co_nutate: 		FB_CO_NUTATE;
	co_aberration:	CO_ABERRATION;
	co_refract:		CO_REFRACT;
	dra1, dra2: LREAL;
	ddec1, ddec2 : LREAL;
END_VAR
VAR CONSTANT
	d2r:	LREAL := PI/180.0;
	h2r:	LREAL := PI/12.0;
	h2d:	LREAL := 15.0;
END_VAR

(* source https://idlastro.gsfc.nasa.gov/ftp/pro/astro/eq2hor.pro 

PURPOSE:
	Convert celestial  (ra-dec) coords to local horizon coords (alt-az).

DESCRIPTION:
This  code calculates horizon (alt,az) coordinates from equatorial
(ra,dec) coords.   It is typically accurate to about 1 arcsecond or better (I
have checked the output against the publicly available XEPHEM software). It
performs precession, nutation, aberration, and refraction corrections.  The
perhaps best thing about it is that it can take arrays as inputs, in all
variables and keywords EXCEPT Lat, lon, and Altitude (the code assumes these
aren't changing), and uses vector arithmetic in every calculation except
when calculating the precession matrices.
*)

ra_ := ra;
dec_ := dec;

tstart := 2000.0;

(* ******************************************************************************
 PRECESS coordinates to current date
 (uses astro lib procedure PRECESS.pro)
*)
J_now := (JD - 2451545.0)/365.25 + 2000.0; // compute current equinox
IF precess THEN
	fbprecess( ra := ra_, dec := dec_, 
	EQUINOX1 := tstart, EQUINOX2 := J_now, 
	ra_precessed =>ra_, dec_precessed => dec_);
END_IF

(******************************************************************************
 calculate NUTATION and ABERRATION Corrections to Ra-Dec 
*)

IF NUTATE THEN
	co_nutate(	jd := jd, 
				ra := ra_, 
				dec := dec_, 
				d_ra => dra1, 
				d_dec => ddec1, 
				eps=>eps, 
				d_psi=>d_psi);
	ra_ := ra_ + dra1/3600.0;
	dec_ := dec_ + ddec1/3600.0;
END_IF

IF ABERRATION THEN	
	co_aberration(	jd := jd, 
					ra := ra_, 
					dec := dec_, 
					d_ra => dra2, 
					d_dec => ddec2, 
					eps := eps);
	ra_ := ra_ + dra2/3600.0;
	dec_ := dec_ + ddec2/3600.0;
END_IF

(***************************************************************************************
Calculate LOCAL MEAN SIDEREAL TIME *)
lmst := ct2lst(lon, jd);  // get LST (in hours) - note:this is independent of time zone  since giving jd
lmst := lmst*h2d ; //convert LMST to degrees (btw, this is the RA of the zenith)
// calculate local APPARENT sidereal time
last := lmst + d_psi *COS(eps*d2r)/3600.0 ; //add correction in degrees

(******************************************************************************
 Find hour angle (in DEGREES) *)
ha := last - ra_;
ha := MODABS(ha, 360.0);

(*******************************************************************************
 Now do the spherical trig to get APPARENT alt,az. *)
hadec2altaz(	ha := ha, 
				dec := dec_, 
				lat := lat, 
				alt => alt, 
				az => az, 
				WS := WS);

(********************************************************************************************
 Make Correction for ATMOSPHERIC REFRACTION
 (use this for visible and radio wavelengths; author is unsure about other wavelengths.
  See the comments in CO_REFRACT for more details.) *)
IF refract THEN 
	co_refract(	old_alt := alt, 
				altitude := altitude, 
				to_observed := TRUE, 
				new_alt => alt);
END_IF

END_FUNCTION_BLOCK

// ---- POUs/FunctionBlocks/FB_HADEC2ALTAZ.TcPOU
FUNCTION_BLOCK FB_HADEC2ALTAZ
VAR_INPUT
	ha,
	dec,
	lat:	LREAL;
	WS:	BOOL := FALSE;
END_VAR
VAR_OUTPUT
	alt,
	az:	LREAL;
END_VAR
VAR
	sh,sd,sl, ch,cd,cl,	x, y, z, radius:	LREAL;
END_VAR
VAR CONSTANT
	d2r :	LREAL := PI/180.0;
END_VAR

(* source https://idlastro.gsfc.nasa.gov/ftp/pro/astro/hadec2altaz.pro *)

sh := SIN(ha*d2r);
ch := COS(ha*d2r);
sd := SIN(dec*d2r);
cd := COS(dec*d2r);
sl := SIN(lat*d2r);
cl := COS(lat*d2r);

x := -ch * cd * sl + sd * cl;
y := -sh * cd;
z := ch * cd * cl + sd * sl;
radius := SQRT(x*x + y*y);

// now get Alt, Az
az := ATAN2(y, x) /d2r;	// was ATAN(y, x)
alt := ATAN2(z, radius) / d2r;

// correct for negative AZ
az := MODABS(az, 360.0);

// convert AZ to West from South, if desired
IF WS THEN 
	az := MODABS(az + 180.0, 360);
END_IF

END_FUNCTION_BLOCK

// ---- POUs/FunctionBlocks/FB_PRECESS2.TcPOU
FUNCTION_BLOCK FB_PRECESS2
VAR_INPUT
	// right ascension in degrees
	ra: LREAL;
	// declination in degrees
	dec: LREAL;
	// starting equinox (J2000)
	equinox1: LREAL;
	// target equinox (J2023 + x)
	equinox2: LREAL;
	// obsolete radian input
	RADIAN:	BOOL := FALSE;
END_VAR
VAR_OUTPUT
	// precessed right ascension
	ra_precessed:	LREAL;
	// precessed declination
	dec_precessed:	LREAL;
END_VAR
VAR
	ra_rad, dec_rad: LREAL;
	dra: LREAL; // in arcsec
	dde: LREAL; // in arcsec
END_VAR
VAR CONSTANT
	deg_to_rad : LREAL := PI/180.0;
	sec_to_rad : LREAL := deg_to_rad/3600.0;
	y100 : LREAL := 23.0/100.0;
END_VAR

ra_rad := ra*deg_to_rad;
dec_rad := dec*deg_to_rad;

IF ABS(dec) < 89.5 THEN
	dra := 46.1244 + 0.0279*y100 + (20.0431-0.0085*y100)*TAN(dec_rad)*SIN(ra_rad);
ELSE
	dra := 0.0;
END_IF

dde := (20.0431 - 0.0085*y100)*COS(ra_rad);

ra_precessed := ra_rad/deg_to_rad + dra/3600.0;
dec_precessed := dec_rad/deg_to_rad + dde/3600.0;

END_FUNCTION_BLOCK

// ---- POUs/FunctionBlocks/TelescopeAxisClass.TcPOU
FUNCTION_BLOCK TelescopeAxisClass
VAR_INPUT
	// enable the axis
	enable: 	BOOL;
	// reset an error
	reset:		BOOL;
	// increase the position
	up:			BOOL;
	// decrease the position
	down:		BOOL;
	// set position of the axis in degrees
	position:	LREAL;
	// set the Velocity of the axis
	velocity:	LREAL;
	// move axis command
	MoveAxis:	BOOL;
	// calibrate the axis
	HomeAxis:	BOOL;
	// enable tracking
	Tracking:	BOOL;
	// stop the Axis
	StopAxis:	BOOL;
END_VAR
VAR_OUTPUT
	// axis is ready to operate
	Ready:			BOOL;
	// drive error condition
	error: 			BOOL;
	// warning condition
	warning:		BOOL;
	// actual position of the elevation axis
	actual_position: 	LREAL;
	// error ID of the elevation axis
	ErrorID: 		UDINT;
	// axis is calibrated
	Calibrated:		BOOL;
	// time to reach target position
	slewtime:		LREAL;
END_VAR
VAR
END_VAR

END_FUNCTION_BLOCK

// ---- POUs/Functions/TEN.TcPOU
FUNCTION TEN : LREAL
VAR_INPUT
	dd,mm,ss: LREAL;
END_VAR
VAR
END_VAR

TEN := dd + (mm/60.0) + (ss/3600.0);

END_FUNCTION

// ---- GlobalTextList.TcGTLO
TEXTLIST GlobalTextList
  272 = 'busy'
  879 = 'Error'
  548 = 'GoHome'
  867 = 'GoTo'
  273 = 'park'
  919 = 'Power'
  120 = 'ready'
  685 = 'Reset'
  777 = 'slew'
  717 = 'sliding'
  155 = 'stopped'
  362 = 'track'
  364 = 'tracking'
END_TEXTLIST

// ---- VISUs/Visualization.TcVIS
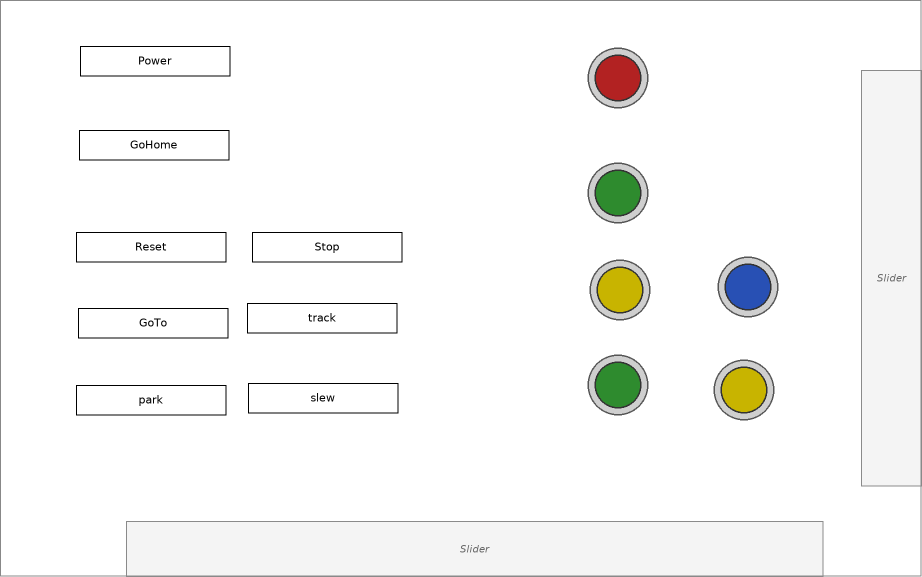
VISUALIZATION Visualization  // 922x577
    RoundedRectangle (80,46 150x30), "Power", colour toggle: TelescopeControl.power
        toggle TelescopeControl.power
    Rectangle (79,130 150x30), "GoHome", colour toggle: TelescopeControl.gohome
        toggle TelescopeControl.gohome
    Lamp1 (583,43 70x70), tooltip "Error", variable: TelescopeControl.error, style: Lamp-Lamp1-Red
    Lamp1 (583,158 70x70), tooltip "ready", variable: TelescopeControl.ready, style: Lamp-Lamp1-Green
    Rectangle (76,232 150x30), "Reset", colour toggle: TelescopeControl.reset
        toggle TelescopeControl.reset
    RoundedRectangle (78,308 150x30), "GoTo", colour toggle: TelescopeControl.goto
        toggle TelescopeControl.goto
    Lamp1 (585,255 70x70), tooltip "sliding", variable: TelescopeControl.sliding, style: Lamp-Lamp1-Yellow
    RoundedRectangle (76,385 150x30), "park", colour toggle: TelescopeControl.park
        toggle TelescopeControl.park
    Lamp1 (583,350 70x70), tooltip "stopped", variable: TelescopeControl.stopped, style: Lamp-Lamp1-Green
    Slider (126,521 697x56), variable: TelescopeControl.rightascension, scale 0..360
    Slider (861,70 61x416), variable: TelescopeControl.declination, scale -90..90
    Lamp1 (713,252 70x70), tooltip "tracking", variable: TelescopeControl.tracking, style: Lamp-Lamp1-Blue
    RoundedRectangle (247,303 150x30), "track", colour toggle: TelescopeControl.track
        toggle TelescopeControl.track
    RoundedRectangle (248,383 150x30), "slew", colour toggle: TelescopeControl.slew
        toggle TelescopeControl.slew
    Lamp1 (709,355 70x70), tooltip "busy", variable: TelescopeControl.busy, style: Lamp-Lamp1-Yellow
    RoundedRectangle (252,232 150x30), "Stop", colour toggle: TelescopeControl.stop
        toggle TelescopeControl.stop
END_VISUALIZATION
